VAR_IN_OUT
	events	: 	ST_ExtController_Events;
	Input	:	ST_PNInput_powerstack;
	Output	:	ST_PNOutput_powerstack;
END_VAR

VAR_INST
	test	:	Real;
END_VAR

//Fill output data
Output.w_Status.0	:=	Monitor.powerstack.Netcontactor.b_NetConFb;
Output.w_Status.1	:=	Monitor.powerstack.b_ACDetected;
Output.w_Status.2	:=	Monitor.powerstack.b_DCDetected;
Output.w_Status.3	:= 	Monitor.powerstack.b_GridTied;
Output.w_Status.4	:=	Monitor.powerstack.b_InverterRunning;
Output.w_Status.5	:=	Monitor.powerstack.b_StartedState;
Output.w_Status.6	:=	Monitor.powerstack.b_ControlEnabled;
Output.w_Status.7	:= 	Monitor.powerstack.b_EcomodeAvailable;
Output.w_Status		:= WordEndian(Output.w_Status);

Output.w_Warnings.0	:=	Monitor.powerstack.Events.b_UndervoltageWarning;
Output.w_Warnings.1	:=	Monitor.powerstack.Events.b_OvervoltageWarning;
Output.w_Warnings.2	:=	Monitor.powerstack.Events.b_overcurrentWarning;
Output.w_Warnings.3	:=	Monitor.powerstack.Events.b_TemperatureWarning OR Monitor.powerstack.Events.b_TemperatureDeviationHigh;
Output.w_Warnings.4	:=	Monitor.powerstack.Events.b_MasterWarning;
Output.w_Warnings.5	:=	Monitor.powerstack.Events.b_SlaveWarning;
Output.w_Warnings.6 := 	Monitor.powerstack.Events.b_GridCodeWarning;
Output.w_Warnings.7 := 	Monitor.powerstack.Netcontactor.events.b_IllegalLeftFieldSelected;
Output.w_Warnings	:= 	WordEndian(Output.w_Warnings);

Output.w_Faults.0	:=	Monitor.powerstack.Events.b_UnderVoltageFault;
Output.w_Faults.1	:=	Monitor.powerstack.Events.b_OverVoltageFault;
Output.w_Faults.2	:=	Monitor.powerstack.Events.b_OvercurrentFault;
Output.w_Faults.3	:=	Monitor.powerstack.Events.b_TemperatureFault;
Output.w_Faults.4	:=	Monitor.powerstack.Events.b_MasterFault;
Output.w_Faults.5	:=	Monitor.powerstack.Events.b_SlaveFault;
Output.w_Faults.6	:=	Monitor.powerstack.Events.b_NetcontactorFault;
//Output.w_Faults.7	:=	monitor.powerstack.Events.b_GridCodeWarning;
Output.w_Faults.8	:=	Monitor.powerstack.Events.b_ShutdownTimeOut OR Monitor.powerstack.Events.b_startupTimeOut;
Output.w_Faults		:= WordEndian(output.w_Faults);

Output.ui_PowerStackStatus			:=  WordEndian(TO_UINT(Monitor.powerstack.e_State));
Output.ui_ACCurrent					:=  RealToUint 	(	In	:= Monitor.powerstack.r_AcCurrent, 		Scale	:=	10);
Output.i_ActivePower				:=  RealToint 	(	In	:= Monitor.powerstack.r_ActivePower, 	Scale	:=	10);
Output.i_ReactivePower 				:= 	RealToint 	(	In	:= Monitor.powerstack.r_ReactivePower, 	Scale	:=	10);
Output.ui_Supplyfrequency 			:=  RealToUint	(	In	:= Monitor.powerstack.r_FrequencyD7, 	Scale	:=	100);
Output.ui_SupplyVoltage				:=  RealToUint 	(	In	:= Monitor.powerstack.r_ACVoltageD7, 	Scale	:=	10);
Output.i_PsetAct 					:=  RealToint 	(	In	:= get.Operation.system.r_Pset, 		Scale	:=	10);
Output.i_QsetAct 					:=  RealToint 	(	In	:= get.Operation.system.r_Qset, 		Scale	:=	10);
Output.i_PFSetAct					:=  RealToUint	( 	In	:= get.Operation.system.r_PFset, 		Scale	:=	10);
Output.ui_LoadPercentage			:=	RealToUint 	( 	IN 	:= Monitor.powerstack.r_LoadPercent, 	Scale	:=	10);
Output.ui_RatedCurrent				:=	RealToUint	( 	In	:= Monitor.powerstack.r_RatedCurrent, 	Scale	:=	10);
Output.ui_RatedPower				:=	RealToUint	( 	In	:= Monitor.powerstack.r_RatedPower, 	Scale	:=	10);
Output.ui_DischargePowerLimit		:= 	RealToUint	( 	In	:= Monitor.powerstack.r_Pmax, 			Scale	:=	10);
Output.ui_ChargePowerLimit			:= 	RealToUint	( 	In	:= ABS(Monitor.powerstack.r_Pmin), 		Scale	:=  10);
Output.ui_ACcurrentLimit			:= 	RealToUint	( 	In	:= Monitor.powerstack.r_ACcurrentLimit, Scale	:=	10);
Output.ui_ApparentPowerLimit		:= 	RealToUint	( 	In	:= Monitor.powerstack.r_Smax, 			Scale	:=	10);
Output.ui_ReactivePowerLimit		:=	RealToUint	(	In  := Monitor.powerstack.r_QMax,			Scale 	:=  10);

//process input data
IF (NOT events.b_HeartbeatFault) THEN
	Input.w_Control := wordEndian(Input.w_Control);
	Get.operation.system.b_PFsetEnable 								:=	Input.w_Control.0;	
	
	IntToReal(	in			:= Input.i_Pset, 
				scale 		:= 10, 
				limitlow	:= -st_params.Limits.r_InverterPowerLimit,
				limithigh	:=	st_params.limits.r_InverterPowerLimit,
    			OutOfRange 	=>	events.b_PsetOutOfRange,
				IgnoreZero 	:= FALSE,
				Out 		:= Get.Operation.system.r_Pset);
				
	IntToReal(	in			:= Input.i_Qset, 
				scale 		:= 10, 
				limitlow	:= -st_params.Limits.r_InverterPowerLimit,
				limithigh	:=	st_params.limits.r_InverterPowerLimit,
    			OutOfRange 	=>	events.b_QsetOutOfRange,
				IgnoreZero 	:= FALSE,
				Out 		:= Get.Operation.system.r_Qset);
	
	IntToReal(	in			:= Input.i_PFset, 
				scale 		:= 100, 
				limitlow	:= -1,
				limithigh	:=	1,
    			OutOfRange 	=>	events.b_PFsetOutOfRange,
				IgnoreZero 	:= TRUE,
				Out 		:= Get.Operation.system.r_PFset);
				
	IF ExternalControlMode > eExternalControlMode.BasicControl THEN
			Settings.MachineParams.system.Powercontroller.SocDroop.enable	:=	Input.w_Control.1;
			Get.SoftSettings.system.b_EcoModeEnable							:= 	Input.w_Control.2;
	
			
		UIntToReal(	in			:= Input.ui_NominalVoltage, 
					scale 		:= 1, 
					limitlow	:= st_params.limits.r_NominalVoltageMin,
					limithigh	:=	st_params.limits.r_NominalVoltageMax,
					OutOfRange 	=>	events.b_NominalVoltageOutOfRange,
					IgnoreZero 	:= TRUE,
					Out 		:= Get.Operation.system.r_NominalVoltage);
		
		UIntToReal(	in			:= Input.ui_NominalFrequency, 
					scale 		:= 100, 
					limitlow	:= st_params.limits.r_NominalFreqMin,
					limithigh	:=	st_params.limits.r_NominalFreqMax,
					OutOfRange 	=>	events.b_NominalFreqOutOfRange,
					IgnoreZero 	:= TRUE,
					Out 		:= Get.Operation.system.r_NominalFrequency);
		
		UIntToReal(	in			:= Input.ui_NominalFrequency, 
					scale 		:= 100, 
					limitlow	:= st_params.limits.r_NominalFreqMin,
					limithigh	:=	st_params.limits.r_NominalFreqMax,
					OutOfRange 	=>	events.b_NominalFreqOutOfRange,
					IgnoreZero 	:= TRUE,
					Out 		:= Get.Operation.system.r_NominalFrequency);
				
		UintToReal(	in			:= Input.ui_FrequencyDroop, 
					scale 		:= 10, 
					limitlow	:=	0, 
					limithigh	:=	st_params.limits.r_DroopMax, 
					OutOfRange 	=>	events.b_FreqDroopOutOfRange,
					IgnoreZero 	:= 	FALSE,
					Out 		:= 	Get.SoftSettings.system.r_FrequencyDroop);
	
		UintToReal(	in			:= 	Input.ui_VoltageDroop, 
					scale 		:= 	10, 
					limitlow	:=	0, 
					limithigh	:=	st_params.limits.r_DroopMax, 
					OutOfRange 	=>	events.b_VoltageDroopOutOfRange,
					IgnoreZero 	:= 	FALSE,
					Out 		:= 	Get.SoftSettings.system.r_VoltageDroop);			
	
//		UintToReal(	in			:= 	Input.ui_PowerRampRate, 
//					scale 		:= 	1, 
//					limitlow	:=	0, 
//					limithigh	:=	st_params.limits.r_PowerRampLimit, 
//					OutOfRange 	=>	events.b_VoltageDroopOutOfRange,
//					IgnoreZero 	:= 	FALSE,
//					Out			:= ?);				
		
				
					
		UintToReal(	in			:= 	Input.ui_SOCDroopUpshiftStart, 
					scale 		:= 	10, 
					limitlow	:=	Settings.MachineParams.system.Powercontroller.SocDroop.SocMinDroopStart, 
					limithigh	:=	get.softsettings.system.r_SocMax, 
					OutOfRange 	=>	events.b_VoltageDroopOutOfRange,
					IgnoreZero 	:= 	TRUE,
					Out 		:= 	Settings.MachineParams.system.Powercontroller.SocDroop.SocMaxDroopStart);
	
		UintToReal(	in			:= 	Input.ui_SOCDroopDownShiftStart, 
					scale 		:= 	10, 
					limitlow	:=	get.softsettings.system.r_SocMin, 
					limithigh	:=	Settings.MachineParams.system.Powercontroller.SocDroop.SocMaxDroopStart, 
					OutOfRange 	=>	events.b_VoltageDroopOutOfRange,
					IgnoreZero 	:= 	TRUE,
					Out 		:= 	Settings.MachineParams.system.Powercontroller.SocDroop.SocMinDroopStart);	
			

	
		CASE input.ui_PowerLimitMode OF
			//	0:	remain 
			1:	get.SoftSettings.system.e_UgridPowerLimitingMode := ePLM.FreqShift;
			2:	get.SoftSettings.system.e_UgridPowerLimitingMode := ePLM.VoltShift;
			3:	get.SoftSettings.system.e_UgridPowerLimitingMode := ePLM.FreqVoltShift;
			4:	get.SoftSettings.system.e_UgridPowerLimitingMode := ePLM.Shutdown;
		END_CASE
		
		UintToReal(	in			:= 	Input.ui_ACCurrentLimit, 
					scale 		:= 	10, 
					limitlow	:=	0, 
					limithigh	:=	monitor.powerstack.r_ACcurrentLimitMax, 
					OutOfRange 	=>	events.b_VoltageDroopOutOfRange,
					IgnoreZero 	:= 	TRUE,
					Out 		:= 	get.SoftSettings.system.r_AMax);
	END_IF
	
ELSE
	//If Heartbeat fails or control is not allowed --> reset Operational values
	// soft settings may remain.
	Get.Operation.system.r_Pset	 :=	0;
	Get.Operation.system.r_Qset	 :=	0;
	Get.Operation.system.r_PFset :=	1;
	Get.Operation.system.r_NominalVoltage := 400;
	get.Operation.system.r_NominalFrequency := 50;
END_IF
END_METHOD

METHOD MapZPT : BOOL
VAR_IN_OUT CONSTANT
	monitor								: ST_System_Monitor;
END_VAR

VAR_IN_OUT
	Output	:	ST_PNOutput_ZPT;
END_VAR

VAR
	HighestTemp	:	Real;
END_VAR


//Fill output data

Output.w_Status.0 	:= 	Monitor.neutraltransformer.b_active;	//not in use
Output.w_Status 	:= WordEndian(Output.w_Status);

Output.w_Warnings.0	:=	Monitor.neutraltransformer.events.b_NeutralCurrentHigh;
Output.w_Warnings.1	:=	Monitor.neutraltransformer.events.b_TemperatureHighPhase[phases.L1] OR 
						Monitor.neutraltransformer.events.b_TemperatureHighPhase[phases.L2] OR 
						Monitor.neutraltransformer.events.b_TemperatureHighPhase[phases.L3];
Output.w_Warnings.2	:=	Monitor.neutraltransformer.events.b_VoltageUnbalanceHigh;
Output.w_Warnings.3	:=	Monitor.neutraltransformer.events.b_NeutralCurrentHigh;
Output.w_warnings 	:= WordEndian(Output.w_Warnings);

Output.w_Errors.0	:=	Monitor.neutraltransformer.events.b_NeutralCurrentTooHigh;
Output.w_Errors.1	:=	Monitor.neutraltransformer.events.b_TemperatureTooHighPhase[phases.L1] OR 
						Monitor.neutraltransformer.events.b_TemperatureTooHighPhase[phases.L2] OR 
						Monitor.neutraltransformer.events.b_TemperatureTooHighPhase[phases.L3];
Output.w_Errors.2	:=	Monitor.neutraltransformer.events.b_VoltageUnbalanceTooHigh;
Output.w_Errors.3	:=	Monitor.neutraltransformer.events.b_NeutralCurrentTooHigh;
Output.w_Errors 	:= WordEndian(Output.w_Errors);

Output.ui_RatedPower:=	RealToUint(in:= Monitor.neutraltransformer.r_ratedPower, Scale:=1); //where to find?
Output.ui_Powerload	:=	RealToUint(in:= Monitor.neutraltransformer.r_Powerload, Scale:=10);

HighestTemp := MAX(Monitor.neutraltransformer.r_TemperaturePhase[0], Monitor.neutraltransformer.r_TemperaturePhase[1], Monitor.neutraltransformer.r_TemperaturePhase[2]);
Output.i_TransformerTemperature	:=	RealToint(in:=HighestTemp, Scale:=10);
END_METHOD

METHOD RealToInt : INT
VAR_INPUT
	In			:	REAL;
	Scale		:	UINT := 10;
END_VAR
IF NOT IsNaN(IN) THEN
	RealToInt := WordEndian(REAL_TO_INT(LIMIT(-32768, In*Scale, 32767)));
END_IF
END_METHOD

METHOD RealToUDINT : UDINT
VAR_INPUT
	In		:	REAL;
	Scale	:	UINT := 10;
END_VAR
IF NOT IsNaN(IN) THEN
	RealToUdint := DwordEndian(REAL_TO_UDINT(LIMIT(0, In*Scale, 16#FFFFFFFF)));
END_IF
END_METHOD

METHOD RealToUint : UINT
VAR_INPUT
	In		:	REAL;
	Scale	:	UINT := 10;
END_VAR
IF NOT IsNaN(IN) THEN
	RealToUint := WordEndian(REAL_TO_UINT(LIMIT(0, In*Scale, 16#FFFF)));
END_IF
END_METHOD

METHOD SetJsonDoc : BOOL
VAR_IN_OUT
	OutputJson       : STRING(2000);
END_VAR


VAR_INST
	fbJson         	: FB_JsonSaxWriter;
  	fbJsonDataType 	: FB_JsonReadWriteDataType;
END_VAR
fbJson.ResetDocument();
fbjson.AddKey('General');
fbJsonDataType.AddJsonValueFromSymbol(fbJson, 'ST_PNOutput_General', SIZEOF(Outputs.General), ADR(Outputs.General));
fbjson.AddKey('Battery');
fbJsonDataType.AddJsonValueFromSymbol(fbJson, 'ST_PNOutput_Battery', SIZEOF(Outputs.Battery), ADR(Outputs.Battery));
fbjson.AddKey('Outputfield');
fbJsonDataType.AddJsonValueFromSymbol(fbJson, 'ST_PNOutput_OutputField', SIZEOF(Outputs.OutputField), ADR(Outputs.OutputField));
fbjson.AddKey('Inputfield');
fbJsonDataType.AddJsonValueFromSymbol(fbJson, 'ST_PNOutput_InputField', SIZEOF(Outputs.InputField), ADR(Outputs.InputField));
fbjson.AddKey('Powerstack');
fbJsonDataType.AddJsonValueFromSymbol(fbJson, 'ST_PNOutput_Powerstack', SIZEOF(Outputs.Powerstack), ADR(Outputs.Powerstack));
fbjson.AddKey('PSB');
fbJsonDataType.AddJsonValueFromSymbol(fbJson, 'ST_PNOutput_PeakShaveBox', SIZEOF(Outputs.PSB), ADR(Outputs.PSB));
fbjson.AddKey('ZPT');
fbJsonDataType.AddJsonValueFromSymbol(fbJson, 'ST_PNOutput_ZPT', SIZEOF(Outputs.ZPT), ADR(Outputs.ZPT));
fbjson.AddKey('InputGen');
fbJsonDataType.AddJsonValueFromSymbol(fbJson, 'ST_PNOutput_Gencontrol', SIZEOF(Outputs.GenControl), ADR(Outputs.GenControl));
fbjson.AddKey('InputGrid');
fbJsonDataType.AddJsonValueFromSymbol(fbJson, 'ST_PNOutput_InputGridControl', SIZEOF(Outputs.InputGridControl), ADR(Outputs.InputGridControl));
fbJson.CopyDocument(OutputJson, SIZEOF(OutputJson));
END_METHOD

METHOD UintToByte : BYTE
VAR_INPUT
	in			:	UINT;
	LimitLow	: 	BYTE;
	LimitHigh	:  	BYTE; 
END_VAR

VAR_OUTPUT
	OutofRange		: BOOL;
END_VAR
OutofRange := ValueOutOfRange(TO_REAL(in), TO_REAL(LimitLow), TO_REAL(LimitHigh));

UintToByte := TO_BYTE(LIMIT(LimitLow, in, LimitHigh));
END_METHOD

METHOD UintToReal : REAL
VAR_INPUT
	in			:	UINT;
	Scale		:	UINT := 1;
	LimitLow	: 	REAL := 0;
	LimitHigh	:  	REAL := 3.402823E+38; 
	IgnoreZero	:	BOOL := FALSE;
END_VAR

VAR_OUTPUT
	OutofRange	: BOOL;
END_VAR

VAR
	r_value			: REAL;
END_VAR

VAR_IN_OUT
	Out	:	REAL;
END_VAR
IF (NOT IgnoreZero) OR (in <> 0) THEN
	r_value	 := UINT_TO_REAL(WordEndian(in))/Scale;
	
	OutofRange := ValueOutOfRange(r_value, LimitLow, LimitHigh);
	Out := LIMIT(LimitLow, r_value, LimitHigh);
END_IF
END_METHOD

METHOD WordEndian : WORD
VAR_INPUT
	IN		: WORD;
END_VAR
IF st_params.b_BigEndian THEN
	WordEndian := HOST_TO_BE16(IN);
ELSE
	WordEndian := IN;
END_IF
END_METHOD

END_FUNCTION_BLOCK

// ---- POUs/MonitoringControl/ExternalControl/FB_ExtControllerTest.TcPOU
FUNCTION_BLOCK FB_ExtControllerTest
//VALUES READ BACK FROM PNCONTROLLER FB
VAR_IN_OUT
	TestVars				: ST_PNTest;
END_VAR

VAR_IN_OUT
	CheckReads					: 	ST_PNOutput;
	//GeneralPLCRead			:	ST_PNOutput_General;
	//BatteryPLCRead 			:	ST_PNOutput_Battery;
	//OutputFieldPLCRead 		:	ST_PNOutput_OutputField;
	//InputFieldPLCRead	 	:	ST_PNOutput_InputField;
	//PowerStackPLCRead	 	:	ST_PNOutput_PowerStack;	
	//PeakShaveBoxPLCRead	 	:	ST_PNOutput_PeakShaveBox;
	//ZPTPLCRead				:	ST_PNOutput_ZPT;
END_VAR

VAR
	WriteReg			:	FB_MBWriteSingleReg;
	ReadRegs			:	FB_MBReadRegs; 
	Ip					: 	STRING := '192.168.1.100';
	Timeout				: 	TIME := T#1S;
	Start				:	BOOL	:= TRUE;
	bComBusy			:	BOOL;
	bComError			:	BOOL;
	errID				:	UDINT;
	
	ComRetryCounter		:	USINT	:= 0; 	
	
	Readbuffer 			: ARRAY [1..100] OF BYTE;
	
	w_heartbeat			: WORD;
END_VAR

VAR
	Reads				:	ST_PNOutput;
	//GeneralPLCCheck			:	ST_PNOutput_General;
	//BatteryPLCCheck 		:	ST_PNOutput_Battery;
	//OutputFieldPLCCheck		:	ST_PNOutput_OutputField;
	//InputFieldPLCCheck	 	:	ST_PNOutput_InputField;
	//PowerStackPLCCheck	 	:	ST_PNOutput_PowerStack;	
	//PeakShaveBoxPLCCheck	:	ST_PNOutput_PeakShaveBox;
	//ZPTPLCCheck				:	ST_PNOutput_ZPT;
END_VAR

IF TestVars.b_CheckMonitoring THEN
	Testvars.b_MonitoringOK := Checkreadings();
END_IF

SetControlValues(TestVars:= Testvars);

METHOD CheckHeartbeat : BOOL

VAR_INST
	index		: WORD;
	
	WriteReg	:	FB_MBWriteSingleReg;
	Addres		: 	WORD	:= 51;
	Value 		:	WORD 	:= 1;
	ComTrigger	:	TON := (PT := TIME#500MS);
END_VAR
ComTrigger(IN:= Start AND NOT ComTrigger.Q AND NOT Readregs.bBusy);

IF value <> Checkreads.general.ui_HeartBeatOut THEN
	value := Checkreads.general.ui_HeartBeatOut;
	CheckHeartbeat := TRUE;
ELSE
	CheckHeartbeat := FALSE;
END_IF

WriteReg(
	sIPAddr := '192.168.1.100',
	nTCPPort := 502,
	nUnitID := 255,//16#FF;
	nMBAddr := Addres,
	nValue := Value,
	tTimeout := T#100MS,
	bExecute := ComTrigger.Q,
	bBusy => bComBusy,
	bError => bComError,
	nErrId => errID,
);
END_METHOD

METHOD CheckReadings : BOOL

VAR_INST
	a_wReadAddress : ARRAY [0..10] OF WORD := [0, 100, 200, 300, 400, 500, 600];
	a_wRegsOnAddres	: ARRAY [0..10] OF WORD := [13, 14, 22, 22, 19, 17, 6];
	readIndex		: WORD;
	cbRead			: UDINT;
	
	ftrigMbBusy		: F_Trig;
	ComTrigger		: TON := (PT := TIME#500MS);
	
	w_DataOK		: WORD;
	b_BufferReady	: BOOL;
END_VAR
ComTrigger(IN:= NOT ComTrigger.Q AND NOT Readregs.bBusy);

ReadRegs(
	sIPAddr	:= IP,
	nTCPPort:= 502,
	nUnitID	:= 255,
	nQuantity:= a_wRegsOnAddres[readindex],
	nMBAddr	:= a_wReadAddress[readindex],
	cbLength:= SIZEOF(Readbuffer),
	pDestAddr:= ADR(Readbuffer),
	bExecute := ComTrigger.Q,
	tTimeOut := Timeout,
	bBusy	=> bComBusy,
	bError	=> bComError,
	nErrID=> errID,
	cbRead => cbRead);

ftrigMbBusy(CLK := bComBusy);
b_BufferReady :=  cbRead = a_wRegsOnAddres[readindex]*2 AND ftrigMbBusy.Q AND NOT bComError;

IF b_BufferReady THEN
	CASE readindex OF
		0: w_DataOK.0 := MEMCMP(pBuf1 := ADR(CheckReads.General), 		pBuf2:= ADR(Readbuffer), n := SIZEOF(CheckReads.General)) = 0;
						 MEMCPY(srcAddr := ADR(Readbuffer), 	destAddr:= ADR(Reads.General), n := SIZEOF(CheckReads.General));
		1: w_DataOK.1 := MEMCMP(pBuf1 := ADR(CheckReads.Battery), 		pBuf2:= ADR(Readbuffer), n := SIZEOF(CheckReads.Battery)) = 0;
						 MEMCPY(srcAddr := ADR(Readbuffer), 	destAddr:= ADR(reads.Battery), n := SIZEOF(CheckReads.Battery));
		2: w_DataOK.2 := MEMCMP(pBuf1 := ADR(CheckReads.OutputField), 	pBuf2:= ADR(Readbuffer), n := SIZEOF(Checkreads.OutputField)) = 0;
						 MEMCPY(srcAddr := ADR(Readbuffer), 	destAddr:= ADR(Reads.OutputField), n := SIZEOF(Checkreads.OutputField));
		3: w_DataOK.3 := MEMCMP(pBuf1 := ADR(Checkreads.InputField) , 	pBuf2:= ADR(Readbuffer), n := SIZEOF(Checkreads.InputField)) = 0;
						 MEMCPY(srcAddr := ADR(Readbuffer), 	destAddr:= ADR(Reads.InputField), n := SIZEOF(Checkreads.InputField));
		4: w_DataOK.4 := MEMCMP(pBuf1 := ADR(Checkreads.PowerStack) , 	pBuf2:= ADR(Readbuffer), n := SIZEOF(Checkreads.PowerStack)) = 0;
						 MEMCPY(srcAddr := ADR(Readbuffer), 	destAddr:= ADR(Reads.PowerStack), n := SIZEOF(Checkreads.PowerStack));
		5: w_DataOK.5 := MEMCMP(pBuf1 := ADR(Checkreads.PSB) , pBuf2:= ADR(Readbuffer), n := SIZEOF(Checkreads.PSB)) = 0;
						 MEMCPY(srcAddr := ADR(Readbuffer), 	destAddr:= ADR(Reads.PSB), n := SIZEOF(Checkreads.PSB));
		6: w_DataOK.6 := MEMCMP(pBuf1 := ADR(Checkreads.ZPT) , 	pBuf2:= ADR(Readbuffer), n := SIZEOF(Checkreads.ZPT)) = 0;
						 MEMCPY(srcAddr := ADR(Readbuffer), 	destAddr:= ADR(Reads.ZPT), n := SIZEOF(Checkreads.ZPT));
	END_CASE
END_IF

IF b_BufferReady THEN
	readIndex := readIndex +1;
END_IF


//Reset index
IF readindex = 7 THEN
	readindex := 0;
END_IF
	
	
CheckReadings := w_DataOK = 127;
END_METHOD

METHOD SetControlValues : BOOL
VAR_IN_OUT
	TestVars				: ST_PNTest;
END_VAR

VAR_INST
	index		: WORD;
	w_control			: WORD;
	
	WriteReg	:	FB_MBWriteSingleReg;
	Addres		: 	WORD	:= 0;
	Value 		:	WORD 	:= 1;
	errID		:	UDINT;
	TransmissionDone 	: 	f_trig;
	ComTrigger	:	Ton := (PT := TIME#200MS);
	ComRetryCounter	:	USINT	:= 0; 
END_VAR
ComTrigger(IN:= NOT ComTrigger.Q AND NOT WriteReg.bBusy);

w_control.0 := testvars.bit_start;
w_control.1 := testvars.bit_stop;
w_control.2 := testvars.bit_shutdown;
w_control.3 := testvars.bit_Systemshutdown;
w_control.4 := testvars.bit_Reset;
w_control.5 := testvars.bit_EMstop;
w_control.6 := testvars.bit_AutoSwitching;
w_control.7 := testvars.bit_TransportMode;
w_control.9 := testvars.bit_AdvancedControl;

CASE (index) OF
	0: Addres := 50; value:= W_Control;
	1: Addres := 453; value:= TO_WORD(testvars.i_Pset);
	2: Addres := 454; value:= TO_WORD(testvars.i_Qset);
	3: Addres := 51; value:= Checkreads.general.ui_HeartBeatOut;
	4: Addres := testvars.w_SetAddress; value:= testvars.w_SetValue;
END_CASE

WriteReg(
	sIPAddr := '192.168.1.100',
	nTCPPort := 502,
	nUnitID := 255,//16#FF;
	nMBAddr := Addres,
	nValue := Value,
	tTimeout := T#100MS,
	bExecute := ComTrigger.Q,
	bBusy => bComBusy,
	bError => bComError,
	nErrId => errID,
);

TransmissionDone(CLK := bComBusy AND NOT bComError);
IF TransmissionDone.Q THEN
	index := index +1;
END_IF

IF index > 4 THEN
	index := 0;
END_IF
END_METHOD

END_FUNCTION_BLOCK

// ---- POUs/Functions-FBs-Programs/_generalFunctions/Scale.TcPOU
FUNCTION Scale : REAL
VAR_INPUT
	r_in	: REAL;
	In_min : REAL;
	In_max : REAL;
	Out_min: REAL;
	Out_max: REAL;
END_VAR

VAR
	r_Temp			: REAL;
	r_inLimited		: REAL;
	r_offset		: REAL;
	r_ratio			: REAL;
END_VAR

IF In_Min < In_Max THEN
	r_inLimited := LIMIT(In_Min, r_in, In_Max);
ELSE
	r_inLimited := LIMIT(In_Max, r_in, In_Min);
END_IF



//IF In_Min < In_Max THEN
	r_offset := r_inLimited - In_Min;
	r_ratio := (Out_Max - Out_Min) / SEL((In_Max - In_Min) =0,(In_Max - In_Min), 1);
	Scale := Out_Min + r_Offset * r_ratio;
//END_IF

END_FUNCTION

// ---- POUs/Functions-FBs-Programs/_generalFunctions/ValueOutOfRange.TcPOU
FUNCTION ValueOutOfRange : BOOL
VAR_INPUT
	r_var				:REAL;
	r_Min				:REAL;
	r_Max				:REAL;
END_VAR

IF r_var >= r_Min AND r_var <= r_Max THEN
	ValueOutOfRange := FALSE;
ELSE
	ValueOutOfRange := TRUE;
END_IF

END_FUNCTION

// ---- POUs/Functions-FBs-Programs/_generalFunctions/IsNaN.TcPOU
FUNCTION IsNaN : BOOL
VAR_INPUT
	IN : REAL;
END_VAR
VAR
	tempdword : DWORD;
	testword : WORD;
END_VAR

tempdword := PDWORD_TO_DWORD(ADR(In));
memcpy(ADR(TestWord), ADR(tempdword) +2, 2);

IsNaN := ((TestWord AND 2#0111111110000000) = 2#0111111110000000);

END_FUNCTION

// ---- POUs/MonitoringControl/FB_TestScripts.TcPOU
FUNCTION_BLOCK FB_TestScripts
VAR_IN_OUT CONSTANT
	monitor								: ST_System_Monitor;
END_VAR
VAR_IN_OUT
	Controlvars			: ST_HMI_Control;
END_VAR

VAR
	b_enable :BOOL := FALSE;
	fbEventLogClient : FB_EventLogClient;
END_VAR

fbEventLogClient.LogEventOnRise(
	ID := 0,
	Trigger := Controlvars.control.b_ActivateSettings,
	eCategory := eEventLogCategory.ReleaseTrigger,
	eSeverity := eEventLogSeverity.Info,
	Message := 'Activate settings trigger received');

CyclicPowerTest(b_enable);

SinusPower(Period := T#10S, offset := 0, Amplitude := 100);

METHOD CapacityTestRoutine : BOOL
VAR_INPUT
	StartCapacityTest	:	BOOL;
	HaltCapacityTest	: 	BOOL;
END_VAR

VAR_INST
	FileOpen	:	FB_FileOpen;
	FileWrite	:	FB_FilePuts;
	FileClose	:	FB_FileClose;
	
	rtrig_FileOpen		:	r_trig;
	rtrig_FileWrite		:	r_trig;
	rtrig_FileClose		:	r_trig;
	
	ftrig_FileOpenDone	:	f_trig;
	rtrig_FileWrite		:	r_trig;
	rtrig_FileClose		:	r_trig;
	
	Filename	:	STRING := 'C:\Users\Administrator\Documents\CapacityTestResult.txt';
	Filehandle	: UINT;
	
	RestPeriod	: 	TIME	:= T#1H;
	TestPowerLevel		:	REAL	:=	200; //200kw
	
	rtrig_starttest		:	r_trig;
	ftrig_filehandler	:	f_trig;
	
	TestStep	:	eCapTestState := eCapTestState.init;
	Substep		:	uint := 0;
	
	bWriteText			:	BOOL;
	Logtext				:	STRING;
END_VAR
rtrig_starttest(clk := StartCapacityTest AND TestStep = eCapTestState.init);

IF HaltCapacityTest THEN
	TestStep := eCapTestState.StopSystem;
END_IF

CASE TestStep OF
	eCapTestState.init:
		IF ftrig_FileOpenDone.Q THEN
			IF NOT fileOpen.bError AND Filehandle > 0 THEN
				TestStep := eCapTestState.WriteSerial;
			ELSE
				HaltCapacityTest := TRUE;
			END_IF
		END_IF
		
		
	eCapTestState.WriteSerial:
		Logtext := Concat(Concat('Capacity test for ePU10 serial: ', settings.Properties.s_SerialNumber), '$0A');
		bWriteText := TRUE;
		IF NOT bWriteText THEN
			TestStep := eCapTestState.WriteNameplateCap;
		END_IF
	
	eCapTestState.WriteNameplateCap:
		Logtext := concat(Concat(Concat('Nameplate Capacity: ', settings.Properties.r_RatedEnergyCapacity), ' kWh'), '$0A');
		bWriteText := TRUE;
		IF NOT bWriteText THEN
			TestStep := eCapTestState.WriteDatetime;
		END_IF
		
	eCapTestState.WriteDatetime:
		Logtext := concat(Concat('Test started: ', TO_STRING(gvl.dt_SystemDateTime)), '$0A');
		bWriteText := TRUE;
		IF NOT bWriteText THEN
			TestStep := eCapTestState.StartSystem;
		END_IF
		
	eCapTestState.StartSystem:
		IF NOT monitor.powerstack.b_GridACdetected OR NOT monitor.powerstack.b_InverterRunning THEN
			Logtext := concat('Test halted: System not running ', '$0A');
			bWriteText := TRUE;
			IF NOT bWriteText THEN
				HaltCapacityTest := TRUE;
			END_IF
		ELSE
			TestStep := eCapTestState.InitialCharge;
			SubStep := 0;
		END_IF
	
	
	eCapTestState.InitialCharge:
		controlvars.Operation.system.r_Pset := -TestPowerLevel;
		controlvars.Operation.system.r_Qset := 0;
		
		IF monitor.system.e_State = eSystemState.Discharging_Only THEN
			controlvars.Operation.system.r_Pset := 0;
			
			CASE substep OF
				0:	Logtext := concat(concat('Initial Charge done at ', TO_STRING(gvl.dt_SystemDateTime)), '$0A');
					bWriteText := TRUE;
					IF NOT bWriteText THEN
						substep := substep+1;
					END_IF
				1:	
					Logtext := concat('SBMU1 voltages: ', TO_STRING(monitor.battery.BatteryInfo.ar_CellVoltage[0]));
					Logtext := concat(Logtext, ', ');
					Logtext := concat(Logtext, TO_STRING(monitor.battery.BatteryInfo.ar_CellVoltage[1]));
					Logtext := concat(Logtext, ', ');
					Logtext := concat(Logtext, TO_STRING(monitor.battery.BatteryInfo.ar_CellVoltage[2]));
					Logtext := concat(Logtext, '$0A');
					bWriteText := TRUE;
					IF NOT bWriteText THEN
						substep := substep+1;
					END_IF
			END_CASE
			Logtext := concat(concat('Initial Charge done at ', TO_STRING(gvl.dt_SystemDateTime)), '$0A');
			bWriteText := TRUE;
			IF NOT bWriteText THEN
				HaltCapacityTest := TRUE;
			END_IF
		END_IF
		
	RestPeriod1:
	DischargeCycle:
	RestPeriod2:
	ChargeCycle:
	RestPeriod3:
	StopSystem:
END_CASE

FileOpen(sPathName := FileName, nMode := FOPEN_MODEWRITE OR FOPEN_MODETEXT, bExecute := rtrig_starttest.q, tTimeout := T#1S, hfile => filehandle);
ftrig_FileOpenDone(clk := FileOpen.bBusy);
FileWrite(hfile := Filehandle, sLine := Logtext, bExecute := rtrig_startwrite.Q, tTimeout := T#2S);
FileClose(hfile := Filehandle, rtrig_CloseFile.Q);
END_METHOD

METHOD CyclicPowerTest : BOOL
VAR_INPUT
	start	: BOOL;
END_VAR
VAR_INST
	ftrigReset	: f_trig;
	rtrigStart	: R_Trig;
	tod_Start	: TOD := TOD#7:00:00.000;
	tod_Stop	: TOD := TOD#18:00:00.000;
	
	timeOK		: BOOL;
	Direction	: INT;
	
	PowerSet	: REAL := 320;
END_VAR
//timeOK := TO_TOD(GVL.dt_SystemDateTime) > tod_start AND TO_TOD(GVL.dt_SystemDateTime) < tod_stop; ; 

rtrigStart(CLK:= start);
IF rtrigStart.Q THEN
	controlvars.operation.system.r_Pset := 200;
END_IF

IF start THEN//AND timeOK THEN
	controlvars.operation.system.r_Qset := -200;
	rtrigStart(CLK:= start);

	IF monitor.battery.BatteryInfo.r_SOCScaled < 10 THEN
		Direction := -1;
	ELSIF monitor.battery.BatteryInfo.r_SOCScaled > 95 THEN
		Direction := 1;
	END_IF
	
	controlvars.operation.system.r_Pset := Direction * PowerSet; 
END_IF

ftrigReset(CLK:= START);
IF ftrigReset.Q THEN 
	controlvars.operation.system.r_Pset := 0;
	controlvars.operation.system.r_Qset := 0;
END_IF
END_METHOD

METHOD SinusPower : REAL
VAR_INPUT
	period			: TIME;
	offset			: REAL;
	Amplitude		: UINT := 300;
END_VAR

VAR_INST
	cycletime : INT := 2;
	i : INT;
	PI : REAL := 3.1415926535897932384626433832795;
	
	samples	 : INT;
	RadperSample : REAL;
	Rad			: REAL;
	
	Q			: REAL;
END_VAR
samples := TO_INT(period) / cycletime;
RadPerSample := 2* PI / samples;

Rad := Rad + RadperSample;

IF RAD >= PI THEN
	RAD := 0;
END_IF

Q := Amplitude * SIN(rad) + offset ;
SinusPower := Q;
END_METHOD

END_FUNCTION_BLOCK

// ---- POUs/Eventlogger/FB_EventLogClient.TcPOU
FUNCTION_BLOCK FB_EventLogClient


VAR_STAT
	fbLoggerStatic	: REFERENCE TO FB_Eventlogger;
	e_objectID			: eObject_id;
END_VAR

METHOD PUBLIC Init : BOOL
VAR_INPUT
	Eventlogger	: REFERENCE TO FB_Eventlogger;
END_VAR
IF __ISVALIDREF(Eventlogger) THEN
	fbLoggerStatic REF= Eventlogger;
	Init := TRUE;
END_IF
END_METHOD

METHOD PUBLIC LogEvent : BOOL
VAR_INPUT
	eCategory	: eEventLogCategory;
	eSeverity	: eEventLogSeverity;
	Message		: STRING;
END_VAR
IF __ISVALIDREF(fbLoggerStatic) THEN
	LogEvent := fbLoggerStatic.PushEvent(
		eCategory := eCategory,
		eSeverity := eSeverity,
		sSourceFB := TO_STRING(e_ObjectID),
		sMessage := Message);
END_IF
END_METHOD

METHOD PUBLIC LogEventOnRise : BOOL
// Each call site must pass a unique ID (0..100) so that every trigger
// gets its own independent R_TRIG slot within this FB instance.
VAR_INPUT
	ID			: BYTE;		// unique index per call site, 0..100 per instance
	Trigger		: BOOL; 
	eCategory	: eEventLogCategory;
	eSeverity	: eEventLogSeverity;
	Message		: STRING;
	objectID	: eObject_id;
END_VAR
VAR_INST
	arTrig		: ARRAY[0..100] OF R_TRIG;
END_VAR
IF ID > 100 THEN RETURN; END_IF
arTrig[ID](CLK := Trigger);
IF arTrig[ID].Q THEN
	LogEventOnRise := LogEvent(eCategory := eCategory, eSeverity := eSeverity, Message := Message);
END_IF
END_METHOD

METHOD ObjectID : BOOL
VAR_INPUT
	IN		: eObject_id;
END_VAR
e_objectID := IN;
END_METHOD

END_FUNCTION_BLOCK

// ---- POUs/Eventlogger/FB_Eventlogger.TcPOU
FUNCTION_BLOCK FB_Eventlogger
VAR_IN_OUT
    stParams : ST_EventLogger_Params;
END_VAR

VAR CONSTANT
    cQueueSize              : UINT := 64;
    cDefaultWriteInterval   : TIME := T#1M;
    cDefaultMaxFileSize     : UDINT := 5000000;
    cDefaultMaxFileCount    : UINT := 5;
    cDefaultFillGrade       : LREAL := 0.9;
    cLogFileName            : STRING(255) := 'C:\PLCUtility\ePU10Log.csv';
END_VAR

VAR
    // Queue
    aQueue              : ARRAY[0..63] OF ST_EventLogEntry;
    nWriteIndex         : UINT;
    nReadIndex          : UINT;
    nQueuedItems        : UINT;
    stCurrentEntry      : ST_EventLogEntry;

    // 4026 Event logging replacement
    // EventLogger sink for dynamic runtime messages
    fbTcEventLogger : FB_TcEventLogger;

    // CSV buffer
    sPendingCsv         : STRING(8191);

    // Timing
    tonWriteInterval    : TON;
    tWriteInterval      : TIME;
    nMaxFileSize        : UDINT;
    nMaxFileCount       : UINT;
    lrMaxFillGrade      : LREAL;
    nRotateThreshold    : UDINT;

    // File handling
    fbFileOpen          : FB_FileOpen;
    fbFileWrite         : FB_FileWrite;
    fbFileClose         : FB_FileClose;

    hFile               : UINT;
    eFileState          : UINT;

    bFileOpenExecute    : BOOL;
    bFileWriteExecute   : BOOL;
    bFileCloseExecute   : BOOL;

    bWritePending       : BOOL;
    bOverwriteOnOpen    : BOOL;

    nActiveFileIndex    : UINT;
    aFileSizes          : ARRAY[0..9] OF UDINT;

    sActiveFileName     : STRING(255);
    nPendingWriteLen    : UDINT;
END_VAR

ApplyParams();
tonWriteInterval(IN := TRUE, PT := tWriteInterval);

WHILE nQueuedItems > 0 DO
	stCurrentEntry := aQueue[nReadIndex];
	nReadIndex := (nReadIndex + 1) MOD cQueueSize;
	nQueuedItems := nQueuedItems - 1;
	// TODO: Load state from previously suspended application

	fbTcEventLogger.SendMessageEx(
		nEventId := GetEventId(stCurrentEntry.eCategory),
		eSeverity := SeverityToTcSeverity(eSeverity := stCurrentEntry.eSeverity),
		sMessage := stCurrentEntry.sMessage);
		
	AppendCsv(stEntry := stCurrentEntry);
END_WHILE

IF tonWriteInterval.Q AND (LEN(sPendingCsv) > 0) THEN
	bWritePending := TRUE;
	tonWriteInterval(IN := FALSE);
END_IF

IF bWritePending THEN
	IF nMaxFileSize > 0 THEN
		IF (aFileSizes[nActiveFileIndex] + TO_UDINT(LEN(sPendingCsv))) >= nRotateThreshold THEN
			nActiveFileIndex := (nActiveFileIndex + 1) MOD nMaxFileCount;
			aFileSizes[nActiveFileIndex] := 0;
			bOverwriteOnOpen := TRUE;
		END_IF
	END_IF
	GetActiveFileName();
	
	CASE eFileState OF
		0:
			bFileOpenExecute := TRUE;
			eFileState := 10;
			
		10:
			fbFileOpen(
				sNetId := '',
				sPathName := sActiveFileName,
				nMode := SEL(bOverwriteOnOpen, FOPEN_MODEAPPEND OR FOPEN_MODETEXT, FOPEN_MODEWRITE OR FOPEN_MODETEXT),
				ePath := PATH_GENERIC,
				bExecute := bFileOpenExecute,
				tTimeout := T#2S,
				hFile => hFile);
			bFileOpenExecute := FALSE;
			
			IF NOT fbFileOpen.bBusy THEN
				IF fbFileOpen.bError THEN
					eFileState := 0;
					bWritePending := FALSE;
				ELSE
					bOverwriteOnOpen := FALSE;
					eFileState := 20;
				END_IF
			END_IF
			
		20:
			nPendingWriteLen := TO_UDINT(LEN(sPendingCsv));
			fbFileWrite(
				sNetId := '',
				hFile := hFile,
				pWriteBuff := ADR(sPendingCsv),
				cbWriteLen := nPendingWriteLen,
				bExecute := bFileWriteExecute,
				tTimeout := T#2S);
			
			IF NOT bFileWriteExecute THEN
				bFileWriteExecute := TRUE;
			ELSE
				bFileWriteExecute := FALSE;
			END_IF
			
			IF NOT fbFileWrite.bBusy THEN
				IF fbFileWrite.bError THEN
					eFileState := 30;
				ELSIF fbFileWrite.cbWrite = nPendingWriteLen THEN
					aFileSizes[nActiveFileIndex] := aFileSizes[nActiveFileIndex] + nPendingWriteLen;
					sPendingCsv := '';
					eFileState := 30;
				END_IF
			END_IF
			
		30:
			fbFileClose(
				sNetId := '',
				hFile := hFile,
				bExecute := bFileCloseExecute,
				tTimeout := T#2S);
			
			IF NOT bFileCloseExecute THEN
				bFileCloseExecute := TRUE;
			ELSE
				bFileCloseExecute := FALSE;
			END_IF
			
			IF NOT fbFileClose.bBusy THEN
				eFileState := 0;
				bWritePending := FALSE;
			END_IF
	END_CASE
END_IF

METHOD PRIVATE AppendCsv : BOOL
VAR_INPUT
	stEntry : ST_EventLogEntry;
END_VAR
VAR
	sLine		: STRING(511);
	sCategory	: STRING(31);
	sSeverity	: STRING(31);
END_VAR
sCategory := CategoryToString(eCategory := stEntry.eCategory);
sSeverity := SeverityToString(eSeverity := stEntry.eSeverity);

sLine := CONCAT(stEntry.sTimestamp, ',');
sLine := CONCAT(sLine, sSeverity);
sLine := CONCAT(sLine, '/');
sLine := CONCAT(sLine, sCategory);
sLine := CONCAT(sLine, ',');
sLine := CONCAT(sLine, stEntry.sSourceFB);
sLine := CONCAT(sLine, ',');
sLine := CONCAT(sLine, stEntry.sMessage);
sLine := CONCAT(sLine, '$0D$0A');

IF (LEN(sPendingCsv) + LEN(sLine)) < SIZEOF(sPendingCsv) THEN
	sPendingCsv := CONCAT(sPendingCsv, sLine);
	AppendCsv := TRUE;
END_IF
END_METHOD

METHOD PRIVATE ApplyParams
VAR_INPUT
END_VAR
tWriteInterval := stParams.LogWriteInterval;
IF tWriteInterval <= T#0S THEN
	tWriteInterval := cDefaultWriteInterval;
END_IF

nMaxFileSize := TO_UDINT(stParams.MaxFileSize);
IF nMaxFileSize = 0 THEN
	nMaxFileSize := cDefaultMaxFileSize;
END_IF

nMaxFileCount := TO_UINT(stParams.MaxFileCount);
IF nMaxFileCount = 0 THEN
	nMaxFileCount := cDefaultMaxFileCount;
ELSIF nMaxFileCount > 10 THEN
	nMaxFileCount := 10;
END_IF

lrMaxFillGrade := TO_LREAL(stParams.MaxFillGrade);
IF lrMaxFillGrade <= 0 THEN
	lrMaxFillGrade := cDefaultFillGrade;
ELSIF lrMaxFillGrade > 1 THEN
	lrMaxFillGrade := 1;
END_IF

nRotateThreshold := TO_UDINT(TO_LREAL(nMaxFileSize) * lrMaxFillGrade);
IF nRotateThreshold = 0 THEN
	nRotateThreshold := nMaxFileSize;
END_IF
END_METHOD

METHOD PRIVATE CategoryToString : STRING
VAR_INPUT
	eCategory : eEventLogCategory;
END_VAR
CASE eCategory OF
	eEventLogCategory.SFCStep:
		CategoryToString := 'SFC_STEP';
	eEventLogCategory.ReleaseTrigger:
		CategoryToString := 'RELEASE_TRIGGER';
	eEventLogCategory.Generic:
		CategoryToString := 'GENERIC';
	eEventLogCategory.Output:
		CategoryToString := 'OUTPUT';
	eEventLogCategory.Input:
		CategoryToString := 'INPUT';
END_CASE
END_METHOD

METHOD PRIVATE GetActiveFileName
VAR_INPUT
END_VAR
IF nActiveFileIndex = 0 THEN
	sActiveFileName := cLogFileName;
ELSE
	sActiveFileName := CONCAT('C:\PLCUtility\ePU10Log_', TO_STRING(nActiveFileIndex));
	sActiveFileName := CONCAT(sActiveFileName, '.csv');
END_IF
END_METHOD

METHOD PRIVATE GetEventId : UDINT
VAR_INPUT
	eCategory : eEventLogCategory;
END_VAR
GetEventId := 10000 + TO_UDINT(eCategory);
END_METHOD

METHOD PUBLIC PushEvent : BOOL
VAR_INPUT
	eCategory	: eEventLogCategory;
	eSeverity	: eEventLogSeverity;
	sSourceFB	: STRING;
	sMessage	: STRING;
END_VAR
VAR
	stNewEntry	: ST_EventLogEntry;
	sTimestamp	: STRING(63);
END_VAR
sTimestamp := CONCAT(GVL.s_SystemDate, ' ');
sTimestamp := CONCAT(sTimestamp, GVL.s_SystemTime);

stNewEntry.sTimestamp := sTimestamp;
stNewEntry.eCategory := eCategory;
stNewEntry.eSeverity := eSeverity;
stNewEntry.sSourceFB := sSourceFB;
stNewEntry.sMessage := sMessage;

IF nQueuedItems >= cQueueSize THEN
	nReadIndex := (nReadIndex + 1) MOD cQueueSize;
	nQueuedItems := nQueuedItems - 1;
END_IF

aQueue[nWriteIndex] := stNewEntry;
nWriteIndex := (nWriteIndex + 1) MOD cQueueSize;
nQueuedItems := nQueuedItems + 1;

PushEvent := TRUE;
END_METHOD

METHOD PRIVATE SeverityToString : STRING
VAR_INPUT
	eSeverity : eEventLogSeverity;
END_VAR
CASE eSeverity OF
	eEventLogSeverity.Warning:
		SeverityToString := 'WARNING';
	eEventLogSeverity.Fault:
		SeverityToString := 'FAULT';
ELSE
	SeverityToString := 'INFO';
END_CASE
END_METHOD

METHOD PRIVATE SeverityToTcSeverity : TcEventSeverity
VAR_INPUT
	eSeverity : eEventLogSeverity;
END_VAR
CASE eSeverity OF
	eEventLogSeverity.Warning:
		SeverityToTcSeverity := TcEventSeverity.Warning;
	eEventLogSeverity.Fault:
		SeverityToTcSeverity := TcEventSeverity.Error;
ELSE
	SeverityToTcSeverity := TcEventSeverity.Info;
END_CASE
END_METHOD

END_FUNCTION_BLOCK

// ---- POUs/MonitoringControl/HMI/HMI.TcPOU
PROGRAM HMI

VAR_IN_OUT CONSTANT
	{ attribute 'TcHmiSymbol.Hide' }
	monitor								: ST_System_Monitor;
	{ attribute 'TcHmiSymbol.Hide' }
	PNcontrolvars						: ST_ExtController_get;
	{ attribute 'TcHmiSymbol.Hide' }
	Iotcontrolvars						: ST_ExtController_get;	
	{ attribute 'TcHmiSymbol.Hide' }
	PLCpersistvars						: ST_PLCPersistentvars;
END_VAR

VAR
	{ attribute 'TcHmiSymbol.ShowRecursively' }
	Monitoringvars		: ST_HMI_Monitor;
	{ attribute 'TcHmiSymbol.ShowRecursively' }
	Controlvars			: ST_HMI_Control;
	{ attribute 'TcHmiSymbol.ShowRecursively' }
	Historizevars		: ST_HMI_Historize;
	{ attribute 'TcHmiSymbol.Show' }
	b_refreshHMIdata			: BOOL;
	{ attribute 'TcHmiSymbol.Show' }
	b_settingschanged			: BOOL;
	{ attribute 'TcHmiSymbol.Show' }
	b_ControlAccess				: BOOL;		
END_VAR

VAR
	t_refreshtime				: TIME:= T#1S;
	ton_refreshtimer			: TON;	
	b_initCycle					: BOOL := TRUE;
	buttons						: FB_HMIButtons;
	rTrigResetPowerSetpoints	: R_TRIG;
	
	//HMI Start/Quit vars
	fbHMIstart : NT_StartProcess;
	b_hmistart	: BOOL := TRUE;
	ton_HmiStart: TON;
	fbTaskKill	: NT_StartProcess;
	b_taskKill	: BOOL;
END_VAR

//hard settings PLC to HMI at init
CopyActSettingsFromPLC(b_initCycle);
b_settingschanged := (MEMCMP(ADR(controlvars.HardSettings), ADR(PLCpersistvars.Hardsettings), SIZEOF(PLCpersistvars.Hardsettings)) <> 0);


//HMI REFRESH SIGNAL
ton_refreshtimer(IN:= NOT ton_refreshtimer.Q, PT:=t_refreshtime);
IF ton_refreshtimer.Q THEN
	 b_refreshHMIdata := NOT b_refreshHMIdata;
END_IF

//Read variables mapping
MapPLCVarsToHMIVars();
//ResetHMIVars when event happens.
ResetHMIvarsOnEvent();
ResetControlvarsOnVariant();

//Set array data AND LINK HMI VARIABLES
SetArraydata(arrays := monitoringvars.Arraydata, b_sync := ton_refreshtimer.Q, init := b_initCycle);


//CALL METHODS AND NESTED FUNCTIONBLOCK
buttons(controlvars := controlvars, monitoringvars := monitoringvars, b_controlaccess := b_controlaccess);
//PSB scheduler function functionaly
GetActiveTimeSlotScheduler(enable:= controlvars.SoftSettings.System.b_EnableSchedule,
	timeslot1 := controlvars.SoftSettings.system.ScheduleTimeSlot1,
	timeslot2 := controlvars.SoftSettings.system.ScheduleTimeSlot2);

b_InitCycle := FALSE;

METHOD ConditionalFormatting 
VAR_IN_OUT
	data : ST_HMI_ConditionalFormatting;
	controls : ST_HMI_control;
END_VAR

VAR
	b_GridTakeover	: BOOL;
	b_inputgenset	: BOOL;
END_VAR
b_GridTakeover := monitor.controlfb.Operation.system.b_GridTakeOverEnable AND monitor.system.GenGridController.e_BreakerMode = eBreakerOperationMode.GridFeedthrough;

IF monitor.controlfb.HardSettings.setup.e_ControlSource = 0 AND
	 NOT Monitor.powerstack.b_InverterGridFormingMode AND Monitor.powerstack.b_StartedState OR b_GridTakeover THEN
		data.b_ShowPset := (NOT monitor.peakshavebox.b_active AND NOT monitor.system.GenGridController.b_active) OR b_GridTakeover;
		data.b_ShowQset := NOT Monitor.controlfb.operation.system.b_PFsetEnable;
		data.b_showPFset := Monitor.controlfb.operation.system.b_PFsetEnable AND monitor.controlfb.HardSettings.setup.e_ControlSource = 0 AND Monitor.controlfb.SoftSettings.setup.e_AcInputType <> eACInputType.Genset;
ELSE
	data.b_ShowPset := FALSE;
	data.b_ShowQset := FALSE;
	data.b_ShowPFset := FALSE;
END_IF

data.b_showPSBData := monitor.system.GenGridController.e_PowerControlMode = ePowercontrolmode.PeakshaveExt;
data.b_ShowInputDisconnect := monitor.system.GenGridController.e_BreakerMode <> eBreakerOperationMode.None;
data.b_ShowModeTransButton := monitor.system.GenGridController.b_ShowModeTrans;

(*monitor.system.GenGridController.b_ModeTransActive OR NOT monitor.system.GenGridController.b_ModeTransInhibit AND 
	monitor.system.GenGridController.e_BreakerMode <> eBreakerOperationMode.GenFeedthrough AND monitor.system.GenGridController.e_BreakerMode <> eBreakerOperationMode.none AND monitor.system.GenGridController.e_BreakerMode <> eBreakerOperationMode.GenIso;

*)
b_inputgenset := monitor.system.GenGridController.e_BreakerMode = eBreakerOperationMode.GenDroop OR
							monitor.system.GenGridController.e_BreakerMode = eBreakerOperationMode.GenFix OR
							monitor.system.GenGridController.e_BreakerMode = eBreakerOperationMode.GenIso;
data.b_ShowShowGensetInfo := b_inputgenset OR monitor.system.GenGridController.b_extGensetMode;
data.b_ShowGenManStartStop := NOT Monitor.controlfb.SoftSettings.inputgenset.b_AutoStartStop AND data.b_ShowShowGensetInfo OR monitor.system.GenGridController.e_GensetStartStop = eGensetstartstop.Start;
data.b_ShowExtgenset := NOT b_inputgenset AND monitor.controlfb.SoftSettings.setup.e_AcInputType <> eAcInputType.Genset;
data.b_ShowGensetHybridMode := monitor.system.GenGridController.e_BreakerMode = eBreakerOperationMode.GenIso AND NOT monitor.system.GenGridController.b_extGensetMode;
END_METHOD

METHOD CopyActSettingsFromPLC : BOOL

VAR_IN_OUT
	init	: BOOL;
END_VAR

VAR
	udi_pointer		: POINTER TO ST_Softsettings;
	b_Onchange 		: BOOL;
END_VAR
IF init THEN
	controlvars.HardSettings := PLCpersistvars.Hardsettings;
	controlvars.SoftSettings := PLCpersistvars.Softsettings;
END_IF
END_METHOD

METHOD PRIVATE DataToHMIArrayFormat
VAR_INPUT
	data								: ST_HMI_Monitor_ArrayDataFormat;
	init								: BOOL;
END_VAR

VAR_IN_OUT
	st_DataOut							: ST_HMIData;
END_VAR
// first cycle only
IF init THEN
	st_DataOut.s_Type := data.s_Type;
	st_DataOut.s_Name := data.s_Name;
	IF data.i_precision <> -1 THEN
		st_DataOut.s_unit := data.s_unit;
	END_IF
	
END_IF


IF data.i_precision = -1 THEN
	st_DataOut.s_Data := data.s_unit;
ELSE
	st_DataOut.s_Data := LREAL_TO_FMTSTR(in:=data.r_Data, iprecision := data.i_precision, bRound := TRUE);
END_IF

IF data.b_warning <> st_DataOut.b_warning THEN
	st_DataOut.b_warning := data.b_warning;
END_IF
END_METHOD

METHOD GetAcInputArrayData : ST_HMI_Monitor_ArrayDataFormat
VAR_IN_OUT CONSTANT
	data : ST_Powermonitor_Inputfield;
END_VAR

VAR_INPUT
	id: INT;
END_VAR
CASE ID OF 
	1: 		GetAcInputArrayData.s_Name:= 'MCCB State';
			GetAcInputArrayData.s_Type:= 'Status';
			GetAcInputArrayData.s_unit:= TO_STRING(monitor.ACswitchgear.b_inputMCCBfb);
	2: 		GetAcInputArrayData.s_Name:= 'MCCB Shunt State';
			GetAcInputArrayData.s_Type:= 'Status';
			GetAcInputArrayData.s_unit:= TO_STRING(monitor.ACswitchgear.b_InputMCCBshuntOK);
	3:		GetAcInputArrayData.s_Name:= 'Apparent Power';
			GetAcInputArrayData.s_Type:= 'AC';
			GetAcInputArrayData.s_Unit:= 'kVA';
			GetAcInputArrayData.i_precision:= 0;
			GetAcInputArrayData.r_Data:= data.ar_ApparentPower[0];
	4:		GetAcInputArrayData.s_Name:= 'Active Power';
			GetAcInputArrayData.s_Type:= 'AC';
			GetAcInputArrayData.s_Unit:= 'kW';
			GetAcInputArrayData.i_precision:= 1;
			GetAcInputArrayData.r_Data:= data.ar_ActivePower[0];
	5:		GetAcInputArrayData.s_Name:= 'Reactive Power';
			GetAcInputArrayData.s_Type:= 'AC';
			GetAcInputArrayData.s_Unit:= 'kvar';
			GetAcInputArrayData.i_precision:= 1;
			GetAcInputArrayData.r_Data:= data.ar_ReactivePower[0];
	6:		GetAcInputArrayData.s_Name:= 'Current';
			GetAcInputArrayData.s_Type:= 'AC';
			GetAcInputArrayData.s_Unit:= 'A';
			GetAcInputArrayData.i_precision:= 1;
			GetAcInputArrayData.r_Data:= data.ar_Current[Phases.AVG];
	7:		GetAcInputArrayData.s_Name:= 'Line Voltage';
			GetAcInputArrayData.s_Type:= 'AC';
			GetAcInputArrayData.s_Unit:= 'VAC';
			GetAcInputArrayData.i_precision:= 1;
			GetAcInputArrayData.r_Data:= data.ar_LineVoltage[phases.AVG];
	8:		GetAcInputArrayData.s_Name:= 'Frequency';
			GetAcInputArrayData.s_Type:= 'AC';
			GetAcInputArrayData.s_Unit:= 'Hz';
			GetAcInputArrayData.i_precision:= 2;
			GetAcInputArrayData.r_Data:= data.ar_Frequency[0];
	9: 		GetAcInputArrayData.s_Name:= 'Power factor';
			GetAcInputArrayData.s_Type:= 'AC';
			GetAcInputArrayData.s_Unit:= '-';
			GetAcInputArrayData.i_precision:= 2;
			GetAcInputArrayData.r_Data:= data.ar_PowerFactor[phases.AVG];
	10:		GetAcInputArrayData.s_Name:= 'Voltage Unbalance';
			GetAcInputArrayData.s_Type:= 'AC';
			GetAcInputArrayData.s_Unit:= '%';
			GetAcInputArrayData.i_precision:= 1;
			GetAcInputArrayData.r_Data:= data.r_VoltageUnbalance;
	11:		GetAcInputArrayData.s_Name:= 'THD';
			GetAcInputArrayData.s_Type:= 'AC';
			GetAcInputArrayData.s_Unit:= '%';
			GetAcInputArrayData.i_precision:= 1;
			GetAcInputArrayData.r_Data:= data.ar_CurrentTHD[phases.AVG];
	12:		GetAcInputArrayData.s_Name:= 'L1';
			GetAcInputArrayData.s_Type:= 'AC Current';
			GetAcInputArrayData.s_Unit:= 'A';
			GetAcInputArrayData.i_precision:= 1;
			GetAcInputArrayData.r_Data:= data.ar_Current[phases.L1];
	13:		GetAcInputArrayData.s_Name:= 'L2';
			GetAcInputArrayData.s_Type:= 'AC Current';
			GetAcInputArrayData.s_Unit:= 'A';
			GetAcInputArrayData.i_precision:= 1;
			GetAcInputArrayData.r_Data:= data.ar_Current[phases.L2];
	14:		GetAcInputArrayData.s_Name:= 'L3';
			GetAcInputArrayData.s_Type:= 'AC Current';
			GetAcInputArrayData.s_Unit:= 'A';
			GetAcInputArrayData.i_precision:= 1;
			GetAcInputArrayData.r_Data:= data.ar_Current[phases.L3];
	15:		GetAcInputArrayData.s_Name:= 'N';
			GetAcInputArrayData.s_Type:= 'AC Current';
			GetAcInputArrayData.s_Unit:= 'A';
			GetAcInputArrayData.i_precision:= 1;
			GetAcInputArrayData.r_Data:= data.ar_Current[phases.N];	
	16:		GetAcInputArrayData.s_Name:= 'L1-L2';
			GetAcInputArrayData.s_Type:= 'AC Linevoltage';
			GetAcInputArrayData.s_Unit:= 'VAC';
			GetAcInputArrayData.i_precision:= 1;
			GetAcInputArrayData.r_Data:= data.ar_LineVoltage[phases.L1];
	17:		GetAcInputArrayData.s_Name:= 'L2-L3';
			GetAcInputArrayData.s_Type:= 'AC Linevoltage';
			GetAcInputArrayData.s_Unit:= 'VAC';
			GetAcInputArrayData.i_precision:= 1;
			GetAcInputArrayData.r_Data:= data.ar_LineVoltage[phases.L2];
	18:		GetAcInputArrayData.s_Name:= 'L3-L1';
			GetAcInputArrayData.s_Type:= 'AC Linevoltage';
			GetAcInputArrayData.s_Unit:= 'VAC';
			GetAcInputArrayData.i_precision:= 1;
			GetAcInputArrayData.r_Data:= data.ar_LineVoltage[phases.L3];
	19:		GetAcInputArrayData.s_Name:= 'L1-N';
			GetAcInputArrayData.s_Type:= 'AC Phasevoltage';
			GetAcInputArrayData.s_Unit:= 'VAC';
			GetAcInputArrayData.i_precision:= 1;
			GetAcInputArrayData.r_Data:= data.ar_PhaseVoltage[phases.L1];	
	20:		GetAcInputArrayData.s_Name:= 'L2-N';
			GetAcInputArrayData.s_Type:= 'AC Phasevoltage';
			GetAcInputArrayData.s_Unit:= 'VAC';
			GetAcInputArrayData.i_precision:= 1;
			GetAcInputArrayData.r_Data:= data.ar_PhaseVoltage[phases.L2];
	21:		GetAcInputArrayData.s_Name:= 'L3-N';
			GetAcInputArrayData.s_Type:= 'AC Phasevoltage';
			GetAcInputArrayData.s_Unit:= 'VAC';
			GetAcInputArrayData.i_precision:= 1;
			GetAcInputArrayData.r_Data:= data.ar_PhaseVoltage[phases.L3];
	22: 	GetAcInputArrayData.s_Name:= 'Contactor state';
			GetAcInputArrayData.s_Type:= 'Status';
			GetAcInputArrayData.s_Unit:= TO_STRING(monitor.ACswitchgear.b_InputContactorfb);
	23: 	GetAcInputArrayData.s_Name:= 'Sync state';
			GetAcInputArrayData.s_Type:= 'Status';
			GetAcInputArrayData.s_Unit:= TO_STRING(monitor.ACswitchgear.b_InputSynchronizerfb);
	24: 	GetAcInputArrayData.s_Name:= 'L1';
			GetAcInputArrayData.s_Type:= 'AC Current 1';
			GetAcInputArrayData.s_Unit:= 'A';
			GetAcInputArrayData.i_precision:= 1;
			GetAcInputArrayData.b_warning := monitor.protections.OvercurrentProtection.Events.Input[1][phases.L1].b_warning;
			GetAcInputArrayData.r_Data:= data.powerlock[1].ar_Current[phases.L1];
	25: 	GetAcInputArrayData.s_Name:= 'L2';
			GetAcInputArrayData.s_Type:= 'AC Current 1';
			GetAcInputArrayData.s_Unit:= 'A';
			GetAcInputArrayData.i_precision:= 1;
			GetAcInputArrayData.b_warning := monitor.protections.OvercurrentProtection.Events.Input[1][phases.L2].b_warning;
			GetAcInputArrayData.r_Data:= data.powerlock[1].ar_Current[phases.L2];
	26: 	GetAcInputArrayData.s_Name:= 'L3';
			GetAcInputArrayData.s_Type:= 'AC Current 1';
			GetAcInputArrayData.s_Unit:= 'A';
			GetAcInputArrayData.i_precision:= 1;
			GetAcInputArrayData.b_warning := monitor.protections.OvercurrentProtection.Events.Input[1][phases.L3].b_warning;
			GetAcInputArrayData.r_Data:= data.powerlock[1].ar_Current[phases.L3];
	27: 	GetAcInputArrayData.s_Name:= 'N';
			GetAcInputArrayData.s_Type:= 'AC Current 1';
			GetAcInputArrayData.s_Unit:= 'A';
			GetAcInputArrayData.i_precision:= 1;
			GetAcInputArrayData.b_warning := monitor.protections.OvercurrentProtection.Events.Input[1][phases.N].b_warning;
			GetAcInputArrayData.r_Data:= data.powerlock[1].ar_Current[phases.N];
	28: 	GetAcInputArrayData.s_Name:= 'L1';
			GetAcInputArrayData.s_Type:= 'AC Current 2';
			GetAcInputArrayData.s_Unit:= 'A';
			GetAcInputArrayData.i_precision:= 1;
			GetAcInputArrayData.b_warning := monitor.protections.OvercurrentProtection.Events.Input[2][phases.L1].b_warning;
			GetAcInputArrayData.r_Data:= data.powerlock[2].ar_Current[phases.L1];
	29: 	GetAcInputArrayData.s_Name:= 'L2';
			GetAcInputArrayData.s_Type:= 'AC Current 2';
			GetAcInputArrayData.s_Unit:= 'A';
			GetAcInputArrayData.i_precision:= 1;
			GetAcInputArrayData.b_warning := monitor.protections.OvercurrentProtection.Events.Input[2][phases.L2].b_warning;
			GetAcInputArrayData.r_Data:= data.powerlock[2].ar_Current[phases.L2];
	30: 	GetAcInputArrayData.s_Name:= 'L3';
			GetAcInputArrayData.s_Type:= 'AC Current 2';
			GetAcInputArrayData.s_Unit:= 'A';
			GetAcInputArrayData.i_precision:= 1;
			GetAcInputArrayData.b_warning := monitor.protections.OvercurrentProtection.Events.Input[2][phases.L3].b_warning;
			GetAcInputArrayData.r_Data:= data.powerlock[2].ar_Current[phases.L3];
	31: 	GetAcInputArrayData.s_Name:= 'N';
			GetAcInputArrayData.s_Type:= 'AC Current 2';
			GetAcInputArrayData.s_Unit:= 'A';
			GetAcInputArrayData.i_precision:= 1;
			GetAcInputArrayData.b_warning := monitor.protections.OvercurrentProtection.Events.Input[2][phases.N].b_warning;
			GetAcInputArrayData.r_Data:= data.powerlock[2].ar_Current[phases.N];
	32: 	GetAcInputArrayData.s_Name:= 'Energy in';                 
			GetAcInputArrayData.s_Type:= 'Energy'; 
			GetAcInputArrayData.s_Unit:= 'kWh';                 
			GetAcInputArrayData.i_precision:= 1;
			GetAcInputArrayData.b_warning := data.r_EnergyConsumed < 0;              
			GetAcInputArrayData.r_Data:= data.r_EnergyConsumed;
	33: 	GetAcInputArrayData.s_Name:= 'Energy out';                 
			GetAcInputArrayData.s_Type:= 'Energy'; 
			GetAcInputArrayData.s_Unit:= 'kWh';                 
			GetAcInputArrayData.i_precision:= 1;
			GetAcInputArrayData.b_warning := data.r_EnergySupplied < 0;              
			GetAcInputArrayData.r_Data:= data.r_EnergySupplied;
	ELSE	
		RETURN;			
END_CASE
END_METHOD

METHOD	GetAcOutputArrayData : ST_HMI_Monitor_ArrayDataFormat
VAR_IN_OUT CONSTANT
	data : ST_Powermonitor_Outputfield;
END_VAR

VAR_INPUT
	id: INT;
END_VAR
CASE ID OF 
	1: 		GetAcOutputArrayData.s_Name:= 'MCCB State';
			GetAcOutputArrayData.s_Type:= 'Status';
			GetAcOutputArrayData.s_Unit:= TO_STRING(monitor.ACswitchgear.b_outputMCCBfb);
	2: 		GetAcOutputArrayData.s_Name:= 'MCCB Shunt State';
			GetAcOutputArrayData.s_Type:= 'Status';
			GetAcOutputArrayData.s_Unit:= TO_STRING(monitor.ACswitchgear.b_outputMCCBshuntOK);
	3:		GetAcOutputArrayData.s_Name:= 'Apparent Power';
			GetAcOutputArrayData.s_Type:= 'AC';
			GetAcOutputArrayData.s_Unit:= 'kVA';
			GetAcOutputArrayData.i_precision:= 0;
			GetAcOutputArrayData.r_Data:= data.ar_ApparentPower[0];
	4:		GetAcOutputArrayData.s_Name:= 'Active Power';
			GetAcOutputArrayData.s_Type:= 'AC';
			GetAcOutputArrayData.s_Unit:= 'kW';
			GetAcOutputArrayData.i_precision:= 1;
			GetAcOutputArrayData.r_Data:= data.ar_ActivePower[0];
	5:		GetAcOutputArrayData.s_Name:= 'Reactive Power';
			GetAcOutputArrayData.s_Type:= 'AC';
			GetAcOutputArrayData.s_Unit:= 'kvar';
			GetAcOutputArrayData.i_precision:= 1;
			GetAcOutputArrayData.r_Data:= data.ar_ReactivePower[0];
	6:		GetAcOutputArrayData.s_Name:= 'Current';
			GetAcOutputArrayData.s_Type:= 'AC';
			GetAcOutputArrayData.s_Unit:= 'A';
			GetAcOutputArrayData.i_precision:= 1;
			GetAcOutputArrayData.r_Data:= data.ar_Current[Phases.AVG];
	7:		GetAcOutputArrayData.s_Name:= 'Line Voltage';
			GetAcOutputArrayData.s_Type:= 'AC';
			GetAcOutputArrayData.s_Unit:= 'VAC';
			GetAcOutputArrayData.i_precision:= 1;
			GetAcOutputArrayData.r_Data:= data.ar_LineVoltage[phases.AVG];
	8:		GetAcOutputArrayData.s_Name:= 'Frequency';
			GetAcOutputArrayData.s_Type:= 'AC';
			GetAcOutputArrayData.s_Unit:= 'Hz';
			GetAcOutputArrayData.i_precision:= 2;
			GetAcOutputArrayData.r_Data:= data.ar_Frequency[0];
	9: 		GetAcOutputArrayData.s_Name:= 'Power factor';
			GetAcOutputArrayData.s_Type:= 'AC';
			GetAcOutputArrayData.s_Unit:= '-';
			GetAcOutputArrayData.i_precision:= 2;
			GetAcOutputArrayData.r_Data:= data.ar_PowerFactor[phases.AVG];
	10:		GetAcOutputArrayData.s_Name:= 'Voltage Unbalance';
			GetAcOutputArrayData.s_Type:= 'AC';
			GetAcOutputArrayData.s_Unit:= '%';
			GetAcOutputArrayData.i_precision:= 1;
			GetAcOutputArrayData.r_Data:= data.r_VoltageUnbalance;
	11:		GetAcOutputArrayData.s_Name:= 'THD';
			GetAcOutputArrayData.s_Type:= 'AC';
			GetAcOutputArrayData.s_Unit:= '%';
			GetAcOutputArrayData.i_precision:= 1;
			GetAcOutputArrayData.r_Data:= data.ar_CurrentTHD[phases.AVG];
	12:		GetAcOutputArrayData.s_Name:= 'L1';
			GetAcOutputArrayData.s_Type:= 'AC Current';
			GetAcOutputArrayData.s_Unit:= 'A';
			GetAcOutputArrayData.i_precision:= 1;
			GetAcOutputArrayData.r_Data:= monitor.powermonitor.outputfield.ar_Current[phases.L1];
	13:		GetAcOutputArrayData.s_Name:= 'L2';                            
			GetAcOutputArrayData.s_Type:= 'AC Current';                    
			GetAcOutputArrayData.s_Unit:= 'A';                            
			GetAcOutputArrayData.i_precision:= 1;                          
			GetAcOutputArrayData.r_Data:= monitor.powermonitor.outputfield.ar_Current[phases.L2];
	14:		GetAcOutputArrayData.s_Name:= 'L3';                            
			GetAcOutputArrayData.s_Type:= 'AC Current';                    
			GetAcOutputArrayData.s_Unit:= 'A';                             
			GetAcOutputArrayData.i_precision:= 1;                          
			GetAcOutputArrayData.r_Data:= monitor.powermonitor.outputfield.ar_Current[phases.L3];
	15:		GetAcOutputArrayData.s_Name:= 'N';                             
			GetAcOutputArrayData.s_Type:= 'AC Current';                    
			GetAcOutputArrayData.s_Unit:= 'A';                            
			GetAcOutputArrayData.i_precision:= 1;                          
			GetAcOutputArrayData.r_Data:= data.ar_Current[phases.N];	
	16:		GetAcOutputArrayData.s_Name:= 'L1-L2';
			GetAcOutputArrayData.s_Type:= 'AC Linevoltage';
			GetAcOutputArrayData.s_Unit:= 'VAC';
			GetAcOutputArrayData.i_precision:= 1;
			GetAcOutputArrayData.r_Data:= data.ar_LineVoltage[phases.L1];
	17:		GetAcOutputArrayData.s_Name:= 'L2-L3';
			GetAcOutputArrayData.s_Type:= 'AC Linevoltage';
			GetAcOutputArrayData.s_Unit:= 'VAC';
			GetAcOutputArrayData.i_precision:= 1;
			GetAcOutputArrayData.r_Data:= data.ar_LineVoltage[phases.L2];
	18:		GetAcOutputArrayData.s_Name:= 'L3-L1';
			GetAcOutputArrayData.s_Type:= 'AC Linevoltage';
			GetAcOutputArrayData.s_Unit:= 'VAC';
			GetAcOutputArrayData.i_precision:= 1;
			GetAcOutputArrayData.r_Data:= data.ar_LineVoltage[phases.L3];
	19:		GetAcOutputArrayData.s_Name:= 'L1-N';
			GetAcOutputArrayData.s_Type:= 'AC Phasevoltage';
			GetAcOutputArrayData.s_Unit:= 'VAC';
			GetAcOutputArrayData.i_precision:= 1;
			GetAcOutputArrayData.r_Data:= data.ar_PhaseVoltage[phases.L1];	
	20:		GetAcOutputArrayData.s_Name:= 'L2-N';
			GetAcOutputArrayData.s_Type:= 'AC Phasevoltage';
			GetAcOutputArrayData.s_Unit:= 'VAC';
			GetAcOutputArrayData.i_precision:= 1;
			GetAcOutputArrayData.r_Data:= data.ar_PhaseVoltage[phases.L2];
	21:		GetAcOutputArrayData.s_Name:= 'L3-N';
			GetAcOutputArrayData.s_Type:= 'AC Phasevoltage';
			GetAcOutputArrayData.s_Unit:= 'VAC';
			GetAcOutputArrayData.i_precision:= 1;
			GetAcOutputArrayData.r_Data:= data.ar_PhaseVoltage[phases.L3];					
	22: 	GetAcOutputArrayData.s_Name:= 'L1';
			GetAcOutputArrayData.s_Type:= 'AC Current 1';
			GetAcOutputArrayData.s_Unit:= 'A';
			GetAcOutputArrayData.i_precision:= 1;
			GetAcOutputArrayData.b_warning := monitor.protections.OvercurrentProtection.Events.Output[1][phases.L1].b_warning;
			GetAcOutputArrayData.r_Data:=  data.powerlock[1].ar_Current[phases.L1];
	23: 	GetAcOutputArrayData.s_Name:= 'L2';                
			GetAcOutputArrayData.s_Type:= 'AC Current 1'; 
			GetAcOutputArrayData.s_Unit:= 'A';                 
			GetAcOutputArrayData.i_precision:= 1;
			GetAcOutputArrayData.b_warning := monitor.protections.OvercurrentProtection.Events.Output[1][phases.L2].b_warning;              
			GetAcOutputArrayData.r_Data:= data.powerlock[1].ar_Current[phases.L2];
	24: 	GetAcOutputArrayData.s_Name:= 'L3';                
			GetAcOutputArrayData.s_Type:= 'AC Current 1'; 
			GetAcOutputArrayData.s_Unit:= 'A';                 
			GetAcOutputArrayData.i_precision:= 1;
			GetAcOutputArrayData.b_warning := monitor.protections.OvercurrentProtection.Events.Output[1][phases.L3].b_warning;              
			GetAcOutputArrayData.r_Data:=  data.powerlock[1].ar_Current[phases.L3];
	25: 	GetAcOutputArrayData.s_Name:= 'N';                 
			GetAcOutputArrayData.s_Type:= 'AC Current 1'; 
			GetAcOutputArrayData.s_Unit:= 'A';                 
			GetAcOutputArrayData.i_precision:= 1;
			GetAcOutputArrayData.b_warning := monitor.protections.OvercurrentProtection.Events.Output[1][phases.N].b_warning;              
			GetAcOutputArrayData.r_Data:= data.powerlock[1].ar_Current[phases.N];
	26: 	GetAcOutputArrayData.s_Name:= 'L1';
			GetAcOutputArrayData.s_Type:= 'AC Current 2';
			GetAcOutputArrayData.s_Unit:= 'A';
			GetAcOutputArrayData.i_precision:= 1;
			GetAcOutputArrayData.b_warning := monitor.protections.OvercurrentProtection.Events.Output[2][phases.L1].b_warning;
			GetAcOutputArrayData.r_Data:=  data.powerlock[2].ar_Current[phases.L1];
	27: 	GetAcOutputArrayData.s_Name:= 'L2';                
			GetAcOutputArrayData.s_Type:= 'AC Current 2'; 
			GetAcOutputArrayData.s_Unit:= 'A';                 
			GetAcOutputArrayData.i_precision:= 1; 
			GetAcOutputArrayData.b_warning := monitor.protections.OvercurrentProtection.Events.Output[2][phases.L2].b_warning;             
			GetAcOutputArrayData.r_Data:=  data.powerlock[2].ar_Current[phases.L2];
	28: 	GetAcOutputArrayData.s_Name:= 'L3';                
			GetAcOutputArrayData.s_Type:= 'AC Current 2'; 
			GetAcOutputArrayData.s_Unit:= 'A';                 
			GetAcOutputArrayData.i_precision:= 1;
			GetAcOutputArrayData.b_warning := monitor.protections.OvercurrentProtection.Events.Output[2][phases.L3].b_warning;              
			GetAcOutputArrayData.r_Data:=  data.powerlock[2].ar_Current[phases.L3];
	29: 	GetAcOutputArrayData.s_Name:= 'N';                 
			GetAcOutputArrayData.s_Type:= 'AC Current 2'; 
			GetAcOutputArrayData.s_Unit:= 'A';                 
			GetAcOutputArrayData.i_precision:= 1;
			GetAcOutputArrayData.b_warning := monitor.protections.OvercurrentProtection.Events.Output[2][phases.N].b_warning;              
			GetAcOutputArrayData.r_Data:=  data.powerlock[2].ar_Current[phases.N];
	30: 	GetAcOutputArrayData.s_Name:= 'L1';
			GetAcOutputArrayData.s_Type:= 'AC Current 3';
			GetAcOutputArrayData.s_Unit:= 'A';
			GetAcOutputArrayData.i_precision:= 1;
			GetAcOutputArrayData.b_warning := monitor.protections.OvercurrentProtection.Events.Output[3][phases.L1].b_warning;
			GetAcOutputArrayData.r_Data:=   data.powerlock[3].ar_Current[phases.L1];
	31: 	GetAcOutputArrayData.s_Name:= 'L2';                
			GetAcOutputArrayData.s_Type:= 'AC Current 3'; 
			GetAcOutputArrayData.s_Unit:= 'A';                 
			GetAcOutputArrayData.i_precision:= 1;     
			GetAcOutputArrayData.b_warning := monitor.protections.OvercurrentProtection.Events.Output[3][phases.L2].b_warning;         
			GetAcOutputArrayData.r_Data:=  data.powerlock[3].ar_Current[phases.L2];
	32: 	GetAcOutputArrayData.s_Name:= 'L3';                
			GetAcOutputArrayData.s_Type:= 'AC Current 3'; 
			GetAcOutputArrayData.s_Unit:= 'A';                 
			GetAcOutputArrayData.i_precision:= 1;    
			GetAcOutputArrayData.b_warning := monitor.protections.OvercurrentProtection.Events.Output[3][phases.L3].b_warning;          
			GetAcOutputArrayData.r_Data:=  data.powerlock[3].ar_Current[phases.L3];
	33: 	GetAcOutputArrayData.s_Name:= 'N';                 
			GetAcOutputArrayData.s_Type:= 'AC Current 3'; 
			GetAcOutputArrayData.s_Unit:= 'A';                 
			GetAcOutputArrayData.i_precision:= 1;
			GetAcOutputArrayData.b_warning := monitor.protections.OvercurrentProtection.Events.Output[3][phases.N].b_warning;              
			GetAcOutputArrayData.r_Data:= data.powerlock[3].ar_Current[phases.N];
	34:		GetAcOutputArrayData.s_Name:= 'Rotation field';
			GetAcOutputArrayData.s_Type:= 'AC';
			GetAcOutputArrayData.s_Unit:= TO_STRING(data.e_ACrotationStatus);
	35: 	GetAcOutputArrayData.s_Name:= 'Energy in';                 
			GetAcOutputArrayData.s_Type:= 'Energy'; 
			GetAcOutputArrayData.s_Unit:= 'kWh';                 
			GetAcOutputArrayData.i_precision:= 1;
			GetAcOutputArrayData.b_warning := data.r_EnergyConsumed < 0;              
			GetAcOutputArrayData.r_Data:= data.r_EnergyConsumed;
	36: 	GetAcOutputArrayData.s_Name:= 'Energy out';                 
			GetAcOutputArrayData.s_Type:= 'Energy'; 
			GetAcOutputArrayData.s_Unit:= 'kWh';                 
			GetAcOutputArrayData.i_precision:= 1;
			GetAcOutputArrayData.b_warning := data.r_EnergySupplied < 0;              
			GetAcOutputArrayData.r_Data:= data.r_EnergySupplied;
ELSE	
		RETURN;
END_CASE
END_METHOD

METHOD GetActiveTimeSlotScheduler
VAR_INPUT
	enable			: BOOL;
END_VAR

VAR_IN_OUT
	timeslot1 : ST_scheduleTimeslot;
	timeslot2 : ST_scheduleTimeslot;
END_VAR

VAR
	w_targetToW1 : WORD; //time of week
	w_targetToW2 : WORD;
	w_CurrentToW : WORD;
	w_CurrentDoW : WORD; 
	w_CurrentToD : WORD; // in minutes\
END_VAR

VAR
	w_MillisInMinute: WORD := 60000;
	w_MinutesInHour	: WORD := 60;
	w_MinutesInDay	: WORD := w_MinutesInHour * 24;
END_VAR
IF enable THEN
	//enable weekly evaluation
	IF timeslot1.usi_DayOfWeek = 0 THEN
		w_CurrentDoW := 0;
		timeslot2.usi_DayOfWeek := 0;
	ELSE
		w_CurrentDoW := F_GetDayOfWeek(IN:=GVL.dt_SystemDateTime);
	END_IF

	w_CurrentToD := TO_WORD(TO_DWORD(TO_TOD(GVL.dt_SystemDateTime))/w_MillisInMinute);
	w_CurrentToW := w_CurrentToD + w_CurrentDoW * w_MinutesInDay;
	w_targetToW1 := Hour_Minute_To_TOW(timeslot1.usi_DayOfWeek,timeslot1.usi_HourOfDay, timeslot1.usi_MinuteOfHour);
	w_targetToW2 := Hour_Minute_To_TOW(timeslot2.usi_DayOfWeek,timeslot2.usi_HourOfDay, timeslot2.usi_MinuteOfHour);
	
	IF w_targetToW1 < w_targetToW2 THEN
		Timeslot1.b_active := w_CurrentToW >= w_targetToW1 AND w_CurrentToW < w_targetToW2;
		Timeslot2.b_active := NOT timeslot1.b_active;
	ELSE
		Timeslot2.b_active := w_CurrentToW >= w_targetToW2 AND w_CurrentToW < w_targetToW1;
		Timeslot1.b_active := NOT timeslot2.b_active;
	END_IF	
ELSE
	Timeslot2.b_active := FALSE;
	Timeslot1.b_active := TRUE;
END_IF
END_METHOD

METHOD GetCoolingData : ST_HMI_Monitor_ArrayDataFormat
VAR_IN_OUT CONSTANT
	data			: ST_CoolingSystem_get;
END_VAR

VAR_INPUT
	id: INT;
END_VAR
CASE ID OF 
	1: 		GetCoolingData.s_Name:= 'Mode';
			GetCoolingData.s_Type:= 'status';
			GetCoolingData.s_unit:= TO_STRING(data.CoolingSystemState);
	2: 		GetCoolingData.s_Name:= 'Heatpump status';
			GetCoolingData.s_Type:= 'status';
			GetCoolingData.s_unit:= TO_STRING(data.HeatPumpStatus);
	3: 		GetCoolingData.s_Name:= 'Coolant pressure';
			GetCoolingData.s_Type:= 'measure';
			GetCoolingData.s_Unit:= 'bar';
			GetCoolingData.i_precision:= 2;
			GetCoolingData.r_data:= data.r_CoolantPressure;
	4: 		GetCoolingData.s_Name:= 'Coolant temperature';
			GetCoolingData.s_Type:= 'measure';
			GetCoolingData.s_Unit:= '°C';
			GetCoolingData.i_precision:= 1;
			GetCoolingData.r_data:= data.r_CoolantTemperature;
	5:		GetCoolingData.s_Name:= 'Enclosure Dewpoint';
			GetCoolingData.s_Type:= 'measure';
			GetCoolingData.s_Unit:= '°C';
			GetCoolingData.i_precision:= 1;
			GetCoolingData.r_Data:= data.r_EnclosureDewpoint;
	ELSE	
		RETURN;			
END_CASE
END_METHOD

METHOD GetDcChargerData : ST_HMI_Monitor_ArrayDataFormat
VAR_IN_OUT CONSTANT
	data : ST_AcDcCharger_get;
END_VAR

VAR_INPUT
	id: INT;
END_VAR
CASE ID OF 
	1: 		GetDcChargerData.s_Name:= 'State';
			GetDcChargerData.s_Type:= 'Status';
			GetDcChargerData.s_unit:= TO_STRING(data.e_SystemStatus);
	2:		GetDcChargerData.s_Name:= 'Line Voltage';
			GetDcChargerData.s_Type:= 'AC';
			GetDcChargerData.s_Unit:= 'Vac';
			GetDcChargerData.i_precision:= 1;
			GetDcChargerData.r_Data:= data.ar_ACvoltage[0];
	3:		GetDcChargerData.s_Name:= 'Active Power';
			GetDcChargerData.s_Type:= 'AC';
			GetDcChargerData.s_Unit:= 'kW';
			GetDcChargerData.i_precision:= 1;
			GetDcChargerData.r_Data:= data.ACmeasurements.ar_ActivePower[0];
	4:		GetDcChargerData.s_Name:= 'Current';
			GetDcChargerData.s_Type:= 'AC';
			GetDcChargerData.s_Unit:= 'A';
			GetDcChargerData.i_precision:= 1;
			GetDcChargerData.r_Data:= data.ACmeasurements.ar_Current[0];
	5:		GetDcChargerData.s_Name:= 'Power';
			GetDcChargerData.s_Type:= 'DC';
			GetDcChargerData.s_Unit:= 'kW';
			GetDcChargerData.i_precision:= 1;
			GetDcChargerData.r_Data:= data.r_DcPower;
	6:		GetDcChargerData.s_Name:= 'Voltage';
			GetDcChargerData.s_Type:= 'DC';
			GetDcChargerData.s_Unit:= 'Vdc';
			GetDcChargerData.i_precision:= 1;
			GetDcChargerData.r_Data:= data.r_DcVoltage;
	7:		GetDcChargerData.s_Name:= 'Current';
			GetDcChargerData.s_Type:= 'DC';
			GetDcChargerData.s_Unit:= 'A';
			GetDcChargerData.i_precision:= 1;
			GetDcChargerData.r_Data:= data.r_DcCurrent;
	8:		GetDcChargerData.s_Name:= 'L1';
			GetDcChargerData.s_Type:= 'P';
			GetDcChargerData.s_Unit:= 'kW';
			GetDcChargerData.i_precision:= 1;
			GetDcChargerData.r_Data:= data.ACmeasurements.ar_ActivePower[phases.L1];
	9:		GetDcChargerData.s_Name:= 'L2';
			GetDcChargerData.s_Type:= 'P';
			GetDcChargerData.s_Unit:= 'kW';
			GetDcChargerData.i_precision:= 1;
			GetDcChargerData.r_Data:= data.ACmeasurements.ar_ActivePower[phases.L2];
	10:		GetDcChargerData.s_Name:= 'L3';
			GetDcChargerData.s_Type:= 'P';
			GetDcChargerData.s_Unit:= 'kW';
			GetDcChargerData.i_precision:= 1;
			GetDcChargerData.r_Data:= data.ACmeasurements.ar_ActivePower[phases.L3];
	11:		GetDcChargerData.s_Name:= 'L1';
			GetDcChargerData.s_Type:= 'Linevoltage';
			GetDcChargerData.s_Unit:= 'Vac';
			GetDcChargerData.i_precision:= 1;
			GetDcChargerData.r_Data:= data.ar_ACvoltage[phases.L1];
	12: 	GetDcChargerData.s_Name:= 'L2';                        
			GetDcChargerData.s_Type:= 'Linevoltage';              
			GetDcChargerData.s_Unit:= 'Vac';                       
			GetDcChargerData.i_precision:= 1;                      
			GetDcChargerData.r_Data:= data.ar_ACvoltage[phases.L2];
	13:		GetDcChargerData.s_Name:= 'L3';                        
			GetDcChargerData.s_Type:= 'Linevoltage';              
			GetDcChargerData.s_Unit:= 'Vac';                       
			GetDcChargerData.i_precision:= 1;                      
			GetDcChargerData.r_Data:= data.ar_ACvoltage[phases.L3];
	ELSE	
		RETURN;			
END_CASE
END_METHOD

METHOD GetDcExtData : ST_HMI_Monitor_ArrayDataFormat
VAR_IN_OUT CONSTANT
	data : ST_DCLink_Get;
END_VAR

VAR_INPUT
	id: INT;
END_VAR
CASE ID OF 
	1: 		GetDcExtData.s_Name:= 'State';
			GetDcExtData.s_Type:= 'Status';
			GetDcExtData.s_unit:= SEL(data.b_DCCouplingState, 'Disconnected', 'Connected');
	2:		GetDcExtData.s_Name:= 'Power';
			GetDcExtData.s_Type:= 'DC';
			GetDcExtData.s_Unit:= 'kW';
			GetDcExtData.i_precision:= 1;
			GetDcExtData.r_Data:= data.Powerdata.Power;
	3:		GetDcExtData.s_Name:= 'Voltage';
			GetDcExtData.s_Type:= 'DC';
			GetDcExtData.s_Unit:= 'Vdc';
			GetDcExtData.i_precision:= 1;
			GetDcExtData.r_Data:= data.Powerdata.Voltage;
	4:		GetDcExtData.s_Name:= 'Current';
			GetDcExtData.s_Type:= 'DC';
			GetDcExtData.s_Unit:= 'A';
			GetDcExtData.i_precision:= 1;
			GetDcExtData.r_Data:= data.Powerdata.Current;
	ELSE	
		RETURN;			
END_CASE
END_METHOD

METHOD GetextcontrolData : ST_HMI_Monitor_ArrayDataFormat
VAR_IN_OUT CONSTANT
	data : ST_ExtController_get;
END_VAR


VAR_INPUT
	id: INT;
END_VAR
CASE ID OF 
	1: 		GetextcontrolData.s_Name:= 'Start';
			GetextcontrolData.s_Type:= 'general';
			GetextcontrolData.s_unit:= TO_STRING(data.control.b_start);
	2: 		GetextcontrolData.s_Name:= 'Shutdown';
			GetextcontrolData.s_Type:= 'general';
			GetextcontrolData.s_unit:= TO_STRING(data.control.b_shutdown);		
	3: 		GetextcontrolData.s_Name:= 'Emstop';
			GetextcontrolData.s_Type:= 'general';
			GetextcontrolData.s_unit:= TO_STRING(data.control.b_EMstop);
	4: 		GetextcontrolData.s_Name:= 'Reset';
			GetextcontrolData.s_Type:= 'general';
			GetextcontrolData.s_unit:= TO_STRING(data.control.b_reset);
	5: 		GetextcontrolData.s_Name:= 'Activate settings';
			GetextcontrolData.s_Type:= 'general';
			GetextcontrolData.s_unit:= TO_STRING(data.control.b_ActivateSettings);
	6: 		GetextcontrolData.s_Name:= 'Automatic switching';
			GetextcontrolData.s_Type:= 'general';
			GetextcontrolData.s_unit:= TO_STRING(data.SoftSettings.system.b_AutomaticSwitching);
	7:		GetextcontrolData.s_Name:= 'Condition mode';
			GetextcontrolData.s_Type:= 'general';
			GetextcontrolData.s_Unit:= TO_STRING(data.SoftSettings.system.b_EnableTransportMode);
	8:		GetextcontrolData.s_Name:= 'Start Dehumid';
			GetextcontrolData.s_Type:= 'general';
			GetextcontrolData.s_Unit:= TO_STRING(data.control.b_startDeHum);
	9:		GetextcontrolData.s_Name:= 'SOC min';
			GetextcontrolData.s_Type:= 'battery';
			GetextcontrolData.s_Unit:= '%';
			GetextcontrolData.i_precision:= 0;
			GetextcontrolData.r_Data:= data.SoftSettings.system.r_SocMin;
			GetextcontrolData.b_warning:= data.events.b_SoCLowLimitOutOfRange;
	10:		GetextcontrolData.s_Name:= 'SOC max';
			GetextcontrolData.s_Type:= 'battery';
			GetextcontrolData.s_Unit:= '%';
			GetextcontrolData.i_precision:= 0;
			GetextcontrolData.r_Data:= data.SoftSettings.system.r_SocMax;
			GetextcontrolData.b_warning:= data.events.b_SoCHighLimitOutOfRange;
	11: 	GetextcontrolData.s_Name:= 'PFset enable';
			GetextcontrolData.s_Type:= 'powerstack';
			GetextcontrolData.s_Unit:= TO_STRING(data.operation.system.b_PFsetEnable);
	13: 	GetextcontrolData.s_Name:= 'Reserved';
			GetextcontrolData.s_Type:= 'powerstack';
			GetextcontrolData.s_Unit:= '-';
	14: 	GetextcontrolData.s_Name:= 'Gridmode';
			GetextcontrolData.s_Type:= 'general';
			GetextcontrolData.b_warning := data.events.b_GridModeValueOutOfRange;
			GetextcontrolData.s_Unit:= TO_STRING(data.SoftSettings.setup.e_Gridmode);
	15: 	GetextcontrolData.s_Name:= 'Powermode';
			GetextcontrolData.s_Type:= 'general';
			GetextcontrolData.b_warning := data.events.b_PowerModeValueOutOfRange;
			GetextcontrolData.s_Unit:= TO_STRING(data.SoftSettings.system.e_UgridPowerMode);
	16:		GetextcontrolData.s_Name:= 'Pset';
			GetextcontrolData.s_Type:= 'powerstack';
			GetextcontrolData.s_Unit:= 'kW';
			GetextcontrolData.i_precision:= 1;
			GetextcontrolData.b_warning := data.events.b_PsetOutOfRange;
			GetextcontrolData.r_Data:= data.Operation.system.r_Pset;
	17:		GetextcontrolData.s_Name:= 'Qset';
			GetextcontrolData.s_Type:= 'powerstack';
			GetextcontrolData.s_Unit:= 'kvar';
			GetextcontrolData.i_precision:= 1;
			GetextcontrolData.b_warning := data.events.b_QsetOutOfRange;
			GetextcontrolData.r_Data:= data.Operation.system.r_Qset;
	18:		GetextcontrolData.s_Name:= 'PFset';
			GetextcontrolData.s_Type:= 'powerstack';
			GetextcontrolData.s_Unit:= '-';
			GetextcontrolData.i_precision:= 2;
			GetextcontrolData.b_warning := data.events.b_PFsetOutOfRange;
			GetextcontrolData.r_Data:= data.Operation.system.r_PFset;
	19:		GetextcontrolData.s_Name:= 'Nom voltage';
			GetextcontrolData.s_Type:= 'powerstack';
			GetextcontrolData.s_Unit:= 'VAC';
			GetextcontrolData.i_precision:= 0;
			GetextcontrolData.b_warning := data.events.b_NominalVoltageOutOfRange;
			GetextcontrolData.r_Data:= data.Operation.system.r_NominalVoltage;
	20:		GetextcontrolData.s_Name:= 'Nom frequency';
			GetextcontrolData.s_Type:= 'powerstack';
			GetextcontrolData.s_Unit:= 'Hz';
			GetextcontrolData.i_precision:= 2;
			GetextcontrolData.b_warning := data.events.b_NominalFreqOutOfRange;
			GetextcontrolData.r_Data:= data.Operation.system.r_NominalFrequency;
	21:		GetextcontrolData.s_Name:= 'Voltage droop';
			GetextcontrolData.s_Type:= 'powerstack';
			GetextcontrolData.s_Unit:= '%';
			GetextcontrolData.i_precision:= 1;
			GetextcontrolData.b_warning := data.events.b_VoltageDroopOutOfRange;
			GetextcontrolData.r_Data:= data.Softsettings.system.r_VoltageDroop;
	22:		GetextcontrolData.s_Name:= 'Frequency droop';
			GetextcontrolData.s_Type:= 'powerstack';
			GetextcontrolData.s_Unit:= '%';
			GetextcontrolData.i_precision:= 1;
			GetextcontrolData.b_warning := data.events.b_FreqDroopOutOfRange;
			GetextcontrolData.r_Data:= data.Softsettings.system.r_FrequencyDroop;
	23:		GetextcontrolData.s_Name:= 'P max';
			GetextcontrolData.s_Type:= 'powerstack';
			GetextcontrolData.s_Unit:= 'kW';
			GetextcontrolData.i_precision:= 1;
			GetextcontrolData.b_warning := data.events.b_PmaxOutOfRange;
			GetextcontrolData.r_Data:= data.Softsettings.system.r_PDischargeLimit;
	24:		GetextcontrolData.s_Name:= 'P min';
			GetextcontrolData.s_Type:= 'powerstack';
			GetextcontrolData.s_Unit:= 'kW';
			GetextcontrolData.i_precision:= 1;
			GetextcontrolData.b_warning := data.events.b_PminOutOfRange;
			GetextcontrolData.r_Data:= data.Softsettings.system.r_PChargeLimit;
	26:		GetextcontrolData.s_Name:= 'AC current limit';
			GetextcontrolData.s_Type:= 'powerstack';
			GetextcontrolData.s_Unit:= 'kvar';
			GetextcontrolData.i_precision:= 1;
			GetextcontrolData.b_warning := data.events.b_AmaxOutOfRange;
			GetextcontrolData.r_Data:= data.Softsettings.system.r_Amax;
	28:		GetextcontrolData.s_Name:= 'Feedin current limit';
			GetextcontrolData.s_Type:= 'PSB';
			GetextcontrolData.s_Unit:= 'A';
			GetextcontrolData.i_precision:= 0;
			GetextcontrolData.b_warning := data.events.b_PSBFeedInLimitOutOfRange;
			GetextcontrolData.r_Data:= data.Softsettings.PSB.setpointTimeslot1.r_FeedInCurrentLimitSoft;
	29:		GetextcontrolData.s_Name:= 'Supply current limit';
			GetextcontrolData.s_Type:= 'PSB';
			GetextcontrolData.s_Unit:= 'A';
			GetextcontrolData.i_precision:= 0;
			GetextcontrolData.b_warning := data.events.b_PSBSupplyLimitOutOfRange;
			GetextcontrolData.r_Data:= data.Softsettings.PSB.setpointTimeslot1.r_SupplyCurrentLimitSoft;
	30:		GetextcontrolData.s_Name:= 'Idle charge power';
			GetextcontrolData.s_Type:= 'PSB';
			GetextcontrolData.s_Unit:= 'kW';
			GetextcontrolData.i_precision:= 1;
			GetextcontrolData.b_warning := data.events.b_PSBIdleChargePowerOutOfRange;
			GetextcontrolData.r_Data:= data.Softsettings.PSB.setpointTimeslot1.r_IdleChargePower;
	31:		GetextcontrolData.s_Name:= 'SOC target';
			GetextcontrolData.s_Type:= 'PSB';
			GetextcontrolData.s_Unit:= '%';
			GetextcontrolData.i_precision:= 0;
			GetextcontrolData.b_warning := data.events.b_PSBSocTargetOutOfRange;
			GetextcontrolData.r_Data:= data.Softsettings.PSB.setpointTimeslot1.r_SocTarget;
	32:		GetextcontrolData.s_Name:= 'Feedin current limit';
			GetextcontrolData.s_Type:= 'input';
			GetextcontrolData.s_Unit:= 'A';
			GetextcontrolData.i_precision:= 0;
			GetextcontrolData.b_warning := data.events.b_FeedInLimitOutOfRange;
			GetextcontrolData.r_Data:= data.Softsettings.inputgrid.setpointTimeslot1.r_FeedInCurrentLimitSoft;
	33:		GetextcontrolData.s_Name:= 'Supply current limit';
			GetextcontrolData.s_Type:= 'input';
			GetextcontrolData.s_Unit:= 'A';
			GetextcontrolData.i_precision:= 0;
			GetextcontrolData.b_warning := data.events.b_SupplyLimitOutOfRange;
			GetextcontrolData.r_Data:= data.Softsettings.inputgrid.setpointTimeslot1.r_SupplyCurrentLimitSoft;
	34:		GetextcontrolData.s_Name:= 'Idle charge power';
			GetextcontrolData.s_Type:= 'input';
			GetextcontrolData.s_Unit:= 'kW';
			GetextcontrolData.i_precision:= 1;
			GetextcontrolData.b_warning := data.events.b_IdleChargePowerOutOfRange;
			GetextcontrolData.r_Data:= data.Softsettings.inputgrid.setpointTimeslot1.r_IdleChargePower;
	35:		GetextcontrolData.s_Name:= 'SOC target';
			GetextcontrolData.s_Type:= 'input';
			GetextcontrolData.s_Unit:= '%';
			GetextcontrolData.i_precision:= 0;
			GetextcontrolData.b_warning := data.events.b_SocTargetOutOfRange;
			GetextcontrolData.r_Data:= data.Softsettings.inputgrid.setpointTimeslot1.r_SocTarget;
	36:		GetextcontrolData.s_Name:= 'AMF';
			GetextcontrolData.s_Type:= 'general';
			GetextcontrolData.s_Unit:= TO_STRING(data.SoftSettings.system.b_AMF);
	37:		GetextcontrolData.s_Name:= 'Contactor Syncclose';
			GetextcontrolData.s_Type:= 'input';
			GetextcontrolData.s_Unit:= TO_STRING(data.Operation.inputgrid.b_SyncClose);
	39:		GetextcontrolData.s_Name:= 'SOC start';
			GetextcontrolData.s_Type:= 'input';
			GetextcontrolData.s_Unit:= '%';
			GetextcontrolData.i_precision:= 0;
			GetextcontrolData.b_warning := data.events.b_SocStartOutOfRange;
			GetextcontrolData.r_Data:= data.Softsettings.inputgenset.setpointTimeslot1.r_SoCStart;
	40:		GetextcontrolData.s_Name:= 'SOC stop';
			GetextcontrolData.s_Type:= 'input';
			GetextcontrolData.s_Unit:= '%';
			GetextcontrolData.i_precision:= 0;
			GetextcontrolData.b_warning := data.events.b_SocStopOutOfRange;
			GetextcontrolData.r_Data:= data.Softsettings.inputgenset.setpointTimeslot1.r_SoCStop;
	41:		GetextcontrolData.s_Name:= 'Overload start';
			GetextcontrolData.s_Type:= 'input';
			GetextcontrolData.s_Unit:= '%';
			GetextcontrolData.i_precision:= 0;
			GetextcontrolData.b_warning := data.events.b_BatOloadStartOutOfRange;
			GetextcontrolData.r_Data:= data.Softsettings.inputgenset.setpointTimeslot1.r_BatteryloadStart;
	42:		GetextcontrolData.s_Name:= 'Overload stop';
			GetextcontrolData.s_Type:= 'input';
			GetextcontrolData.s_Unit:= '%';
			GetextcontrolData.i_precision:= 0;
			GetextcontrolData.b_warning := data.events.b_BatOloadStopOutOfRange;
			GetextcontrolData.r_Data:= data.Softsettings.inputgenset.setpointTimeslot1.r_BatteryloadStop;
	43:		GetextcontrolData.s_Name:= 'Manual start';
			GetextcontrolData.s_Type:= 'input';
			GetextcontrolData.s_Unit:= TO_STRING(data.Operation.genset.b_ManualStart);
	44: 	GetextcontrolData.s_Name:= 'Heartbeat';
			GetextcontrolData.s_Type:= 'general';
			GetextcontrolData.s_unit:= TO_STRING(data.ui_Heartbeat);
			GetextControldata.b_warning := data.events.b_HeartbeatFault;
	ELSE	
		RETURN;			
END_CASE
END_METHOD

METHOD	GetGensetData : ST_HMI_Monitor_ArrayDataFormat
VAR_IN_OUT CONSTANT
	data : ST_Genset_get;
END_VAR

VAR_INPUT
	id: INT;
END_VAR

VAR
	modestring : STRING;
	RunningString : STRING;
END_VAR
CASE ID OF 
	1: 		GetGensetData.s_Name:= 'Breaker state';
			GetGensetData.s_Type:= 'Status';
			GetGensetData.s_Unit:= SEL(data.bGenBreakerClosed, 'OPEN', 'CLOSED');
	2: 		GetGensetData.s_Name:= 'Sync state';
			GetGensetData.s_Type:= 'Status';
			GetGensetData.s_Unit:= TO_STRING(data.bMainBreakerClosed);
	3:		GetGensetData.s_Name:= 'Apparent Power';
			GetGensetData.s_Type:= 'AC';
			GetGensetData.s_Unit:= 'kVA';
			GetGensetData.i_precision:= 0;
			GetGensetData.r_Data:= data.ar_ApparentPower[0];
	4:		GetGensetData.s_Name:= 'Active Power';
			GetGensetData.s_Type:= 'AC';
			GetGensetData.s_Unit:= 'kW';
			GetGensetData.i_precision:= 1;
			GetGensetData.r_Data:= data.ar_ActivePower[0];
	5:		GetGensetData.s_Name:= 'Reactive Power';
			GetGensetData.s_Type:= 'AC';
			GetGensetData.s_Unit:= 'kvar';
			GetGensetData.i_precision:= 1;
			GetGensetData.r_Data:= data.ar_ReactivePower[0];
	6:		GetGensetData.s_Name:= 'Current';
			GetGensetData.s_Type:= 'AC';
			GetGensetData.s_Unit:= 'A';
			GetGensetData.i_precision:= 1;
			GetGensetData.r_Data:= data.ar_Current[0];
	7:		GetGensetData.s_Name:= 'Line Voltage';
			GetGensetData.s_Type:= 'AC';
			GetGensetData.s_Unit:= 'VAC';
			GetGensetData.i_precision:= 1;
			GetGensetData.r_Data:= data.ar_LineVoltage[0];
	8:		GetGensetData.s_Name:= 'Phase Voltage';
			GetGensetData.s_Type:= 'AC';
			GetGensetData.s_Unit:= 'VAC';
			GetGensetData.i_precision:= 1;
			GetGensetData.r_Data:= data.ar_PhaseVoltage[0];
	9:		GetGensetData.s_Name:= 'Frequency';
			GetGensetData.s_Type:= 'AC';
			GetGensetData.s_Unit:= 'Hz';
			GetGensetData.i_precision:= 2;
			GetGensetData.r_Data:=  data.ar_Frequency[0];
	10: 	GetGensetData.s_Name:= 'Power factor';
			GetGensetData.s_Type:= 'AC';
			GetGensetData.s_Unit:= '-';
			GetGensetData.i_precision:= 2;
			GetGensetData.r_Data:=  data.ar_Powerfactor[0];
	11:		GetGensetData.s_Name:= 'L1';
			GetGensetData.s_Type:= 'AC Current';
			GetGensetData.s_Unit:= 'A';
			GetGensetData.i_precision:= 1;
			GetGensetData.r_Data:= data.ar_Current[1];
	12:		GetGensetData.s_Name:= 'L2';
			GetGensetData.s_Type:= 'AC Current';
			GetGensetData.s_Unit:= 'A';
			GetGensetData.i_precision:= 1;
			GetGensetData.r_Data:= data.ar_Current[2];
	13:		GetGensetData.s_Name:= 'L3';
			GetGensetData.s_Type:= 'AC Current';
			GetGensetData.s_Unit:= 'A';
			GetGensetData.i_precision:= 1;
			GetGensetData.r_Data:= data.ar_Current[3];
	14:		IF data.bFixedPowerActive THEN
				modestring := 'Fixed Power ';
			ELSIF data.bIslandModeActive THEN
				modestring := 'Island ';
			ELSIF data.bMainsFailure THEN
				modestring := 'Mains Failure ';
			END_IF
			RunningString := SEL(data.bGenRunning, 'Off','Running');
			GetGensetData.s_Name:= 'Mode';
			GetGensetData.s_Type:= 'Status';
			GetGensetData.s_Unit:= CONCAT(ModeString, RunningString);
ELSE	
		RETURN;
END_CASE
END_METHOD

METHOD GetHeatpumpData :  ST_HMI_Monitor_ArrayDataFormat
VAR_IN_OUT CONSTANT
	data			: ST_Heatpump_get;
END_VAR

VAR_INPUT
	id: INT;
END_VAR
CASE ID OF 
	1: 		GetHeatpumpData.s_Name:= 'State';
			GetHeatpumpData.s_Type:= 'status';
			GetHeatpumpData.s_unit:= TO_STRING(data.HeatPumpState);
	2: 		GetHeatpumpData.s_Name:= 'Operating hours';
			GetHeatpumpData.s_Type:= 'status';
			GetHeatpumpData.s_unit:= TO_STRING(data.HeatpumpData.i_OperatingHours);
	3: 		GetHeatpumpData.s_Name:= 'Setpoint';
			GetHeatpumpData.s_Type:= 'data';
			GetHeatpumpData.s_Unit:= '°C';
			GetHeatpumpData.i_precision:= 1;
			GetHeatpumpData.r_data:= data.Setpoint;
	4: 		GetHeatpumpData.s_Name:= 'Inlet water temp';
			GetHeatpumpData.s_Type:= 'data';
			GetHeatpumpData.s_Unit:= '°C';
			GetHeatpumpData.i_precision:= 1;
			GetHeatpumpData.r_data:= data.HeatpumpData.r_InletWaterTemp;
	5: 		GetHeatpumpData.s_Name:= 'Outlet water temp';
			GetHeatpumpData.s_Type:= 'data';
			GetHeatpumpData.s_Unit:= '°C';
			GetHeatpumpData.i_precision:= 1;
			GetHeatpumpData.r_data:= data.HeatpumpData.r_OutletWaterTemp;
	6: 		GetHeatpumpData.s_Name:= 'Comp input temp';
			GetHeatpumpData.s_Type:= 'data';
			GetHeatpumpData.s_Unit:= '°C';
			GetHeatpumpData.i_precision:= 1;
			GetHeatpumpData.r_data:= data.HeatpumpData.r_CompInputTemp;
	7: 		GetHeatpumpData.s_Name:= 'Comp output temp';
			GetHeatpumpData.s_Type:= 'data';
			GetHeatpumpData.s_Unit:= '°C';
			GetHeatpumpData.i_precision:= 1;
			GetHeatpumpData.r_data:= data.HeatpumpData.r_CompOutputTemp;
	8: 		GetHeatpumpData.s_Name:= 'Outdoor temp';
			GetHeatpumpData.s_Type:= 'data';
			GetHeatpumpData.s_Unit:= '°C';
			GetHeatpumpData.i_precision:= 1;
			GetHeatpumpData.r_data:= data.HeatpumpData.r_OutdoorTemp;
	9: 		GetHeatpumpData.s_Name:= 'Low pressure';
			GetHeatpumpData.s_Type:= 'data';
			GetHeatpumpData.s_Unit:= 'bar';
			GetHeatpumpData.i_precision:= 1;
			GetHeatpumpData.r_data:= data.HeatpumpData.r_LowPressure;
	10: 	GetHeatpumpData.s_Name:= 'High pressure';
			GetHeatpumpData.s_Type:= 'data';
			GetHeatpumpData.s_Unit:= 'bar';
			GetHeatpumpData.i_precision:= 1;
			GetHeatpumpData.r_data:= data.HeatpumpData.r_HighPressure;
	11: 	GetHeatpumpData.s_Name:= 'Water flowrate';
			GetHeatpumpData.s_Type:= 'data';
			GetHeatpumpData.s_Unit:= 'L/s';
			GetHeatpumpData.i_precision:= 1;
			GetHeatpumpData.r_data:= data.HeatpumpData.ui_WaterFlowRate;
	12: 	GetHeatpumpData.s_Name:= 'Defrosting';
			GetHeatpumpData.s_Type:= 'status';
			GetHeatpumpData.s_Unit:= SEL(data.HeatpumpData.b_DefrostingActive, 'Active', 'Inactive');
	14: 	GetHeatpumpData.s_Name:= 'Pump speed';
			GetHeatpumpData.s_Type:= 'data';
			GetHeatpumpData.s_Unit:= '%';
			GetHeatpumpData.i_precision:= 1;
			GetHeatpumpData.r_data:= data.HeatpumpData.r_PumpSpeedPCT;
	15: 	GetHeatpumpData.s_Name:= 'Fan speed';
			GetHeatpumpData.s_Type:= 'data';
			GetHeatpumpData.s_Unit:= '%';
			GetHeatpumpData.i_precision:= 1;
			GetHeatpumpData.r_data:= data.HeatpumpData.r_FanSpeedPCT;
ELSE	
		RETURN;			
END_CASE
END_METHOD

METHOD GetMBMUData : ST_HMI_Monitor_ArrayDataFormat
VAR_IN_OUT CONSTANT
	data 			: st_BMS_BatterySummary;
END_VAR

VAR_INPUT
	id: INT;
END_VAR
CASE ID OF 
	1: 		GetMBMUData.s_Name:= 'Status';
			GetMBMUData.s_Type:= 'status';
			GetMBMUData.s_unit:= TO_STRING(data.e_BMS_Status);
	2: 		GetMBMUData.s_Name:= 'Power-on status';
			GetMBMUData.s_Type:= 'status';
			GetMBMUData.s_unit:= TO_STRING(data.e_BMS_PowerOnStatus);
	3:		GetMBMUData.s_Name:= 'Voltage';
			GetMBMUData.s_Type:= 'power';
			GetMBMUData.s_Unit:= 'VDC';
			GetMBMUData.i_precision:= 1;
			GetMBMUData.r_Data:= data.r_SystemVoltage;
	4:		GetMBMUData.s_Name:= 'Current';
			GetMBMUData.s_Type:= 'power';
			GetMBMUData.s_Unit:= 'A';
			GetMBMUData.i_precision:= 1;
			GetMBMUData.r_Data:= data.r_SystemCurrent;
	5:		GetMBMUData.s_Name:= 'Power';
			GetMBMUData.s_Type:= 'power';
			GetMBMUData.s_Unit:= 'kW';
			GetMBMUData.i_precision:= 1;
			GetMBMUData.r_Data:= data.r_SystemPower;
	6:		GetMBMUData.s_Name:= 'Max charge current';
			GetMBMUData.s_Type:= 'limit';
			GetMBMUData.s_Unit:= 'A';
			GetMBMUData.i_precision:= 1;
			GetMBMUData.r_Data:= data.r_MaxChargeCurrentAllowed;
	7:		GetMBMUData.s_Name:= 'Max discharge current';
			GetMBMUData.s_Type:= 'limit';
			GetMBMUData.s_Unit:= 'A';
			GetMBMUData.i_precision:= 1;
			GetMBMUData.r_Data:= data.r_MaxDischargeCurrentAllowed;
	8:		GetMBMUData.s_Name:= 'Max charge power';
			GetMBMUData.s_Type:= 'limit';
			GetMBMUData.s_Unit:= 'kW';
			GetMBMUData.i_precision:= 1;
			GetMBMUData.r_Data:= data.r_MaxChargePowerAllowed;
	9: 		GetMBMUData.s_Name:= 'Max discharge power';
			GetMBMUData.s_Type:= 'limit';
			GetMBMUData.s_Unit:= 'kW';
			GetMBMUData.i_precision:= 1;
			GetMBMUData.r_Data:= data.r_MaxDischargePowerAllowed;
	10:		GetMBMUData.s_Name:= 'Charge SOE';
			GetMBMUData.s_Type:= 'energy';
			GetMBMUData.s_Unit:= '%';
			GetMBMUData.i_precision:= 0;
			GetMBMUData.r_Data:= data.r_ChargeSOE;
	11:		GetMBMUData.s_Name:= 'Discharge SOE';                       
			GetMBMUData.s_Type:= 'energy';                       
			GetMBMUData.s_Unit:= '%';                               
			GetMBMUData.i_precision:= 0;                              
			GetMBMUData.r_Data:= data.r_DischargeSOE;
//	12:		GetMBMUData.s_Name:= 'Total charge energy';                       
//			GetMBMUData.s_Type:= 'energy';                       
//			GetMBMUData.s_Unit:= 'kWh';                               
//			GetMBMUData.i_precision:= 0;                              
//			GetMBMUData.r_Data:= data.r_HistAccChargeEnergy;
//	13:		GetMBMUData.s_Name:= 'Total discharge energy';                         
//			GetMBMUData.s_Type:= 'energy';                                 
//			GetMBMUData.s_Unit:= 'kWh';                                         
//			GetMBMUData.i_precision:= 0;                                        
//			GetMBMUData.r_Data:= data.r_HistAccDischargeEnergy;
			
	14:		GetMBMUData.s_Name:= 'Remaining charge energy';                         
			GetMBMUData.s_Type:= 'energy';                                 
			GetMBMUData.s_Unit:= 'kWh';                                         
			GetMBMUData.i_precision:= 0;                                        
			GetMBMUData.r_Data:= data.r_RemainingChargeEnergy;
	15:		GetMBMUData.s_Name:= 'Remaining discharge energy';                         
			GetMBMUData.s_Type:= 'energy';                                 
			GetMBMUData.s_Unit:= 'kWh';                                         
			GetMBMUData.i_precision:= 0;                                        
			GetMBMUData.r_Data:= data.r_RemainingDischargeEnergy;	
	16:		GetMBMUData.s_Name:= 'Max allowed voltage';                         
			GetMBMUData.s_Type:= 'limit';                                 
			GetMBMUData.s_Unit:= 'VDC';                                         
			GetMBMUData.i_precision:= 1;                                        
			GetMBMUData.r_Data:= data.r_MaxSystemVoltageAllowed;	
	17:		GetMBMUData.s_Name:= 'Min allowed voltage';                                     
			GetMBMUData.s_Type:= 'limit';                                     
			GetMBMUData.s_Unit:= 'VDC';                                             
			GetMBMUData.i_precision:= 1;                                            
			GetMBMUData.r_Data:= data.r_MinSystemVoltageAllowed;
			GetMBMUData.s_Type:= 'cell';                                        
			GetMBMUData.s_Unit:= 'VDC';                                                
			GetMBMUData.i_precision:= 2;                                               
			GetMBMUData.r_Data:= data.ar_CellVoltage[2];
	18:		GetMBMUData.s_Name:= 'SOH';
			GetMBMUData.s_Type:= 'status';
			GetMBMUData.s_Unit:= '%';
			GetMBMUData.i_precision:= 1;
			GetMBMUData.r_Data:= data.r_SOH;	
	19:		GetMBMUData.s_Name:= 'SOC actual';                          
			GetMBMUData.s_Type:= 'status';                  
			GetMBMUData.s_Unit:= '%';                            
			GetMBMUData.i_precision:= 1;                         
			GetMBMUData.r_Data:= data.r_SOC;
	20:		GetMBMUData.s_Name:= 'Cycle count';                          
			GetMBMUData.s_Type:= 'status';                                          
			GetMBMUData.s_unit:= TO_STRING(data.ui_CycleCount);
	ELSE	
		RETURN;			
END_CASE
END_METHOD

METHOD GetPowerModuleArrayData : ST_HMI_Monitor_ArrayDataFormat
VAR_IN_OUT CONSTANT
	data		: ST_Powermodule_get;
END_VAR

